// TIA Portal V16 export
// export: Created 2024-08-19T08:04:42.5186365Z, ExportSetting WithDefaults, DisplayName Totally Integrated Automation Portal, DisplayVersion V16, DisplayName TIA Portal Version Control Interface, DisplayVersion V16, DisplayName TIA Portal Openness, DisplayVersion V16, DisplayName STEP 7 Professional, DisplayVersion V16, DisplayName STEP 7 Safety, DisplayVersion V16, DisplayName WinCC Professional, DisplayVersion V16
DATA_BLOCK "DB00801_St_ConstAiRawData"   // DB801
TITLE = Static DB [SYSTEM CONSTANTS] — Analog Input Card Types, Ranges and Coefficients
{ S7_Optimized_Access := 'TRUE' }
AUTHOR : M_Gledhill
FAMILY : SysConstants
NAME : St_ConstAiRawData
VERSION : 1.0
// PRACTICAL SERIES AUTOMATION LIBRARY (PAL)   —   COPYRIGHT 2020 – M. GLEDHILL (MIT LICENCE)
//                   ———— ◆ ————
// FULL ONLINE DOCUMENTATION IS AVAILABLE AT: https://practicalseries.com/2001-pal/index.html
// stored: AutoNumber false, DBAccessibleFromOPCUA true, IsOnlyStoredInLoadMemory false, IsRetainMemResEnabled false, IsWriteProtectedInAS false, MemoryReserve 100
   VAR
      _DB_Header { ExternalAccessible := 'False'; ExternalVisible := 'False'; ExternalWritable := 'False'} : Array[0..79] of Bool;   // Static DB [SYSTEM CONSTANTS] — Analog Input Card Types, Ranges and Coefficients
      __________0000_0 { ExternalAccessible := 'False'; ExternalVisible := 'False'; ExternalWritable := 'False'} : Bool := false;
      __________0000_1 { ExternalAccessible := 'False'; ExternalVisible := 'False'; ExternalWritable := 'False'} : Bool := false;
      revInfo { ExternalWritable := 'False'} : "UT01000_St_SysRevision";
      __________0010_0 { ExternalAccessible := 'False'; ExternalVisible := 'False'; ExternalWritable := 'False'} : Bool := false;
      __________0010_1 { ExternalAccessible := 'False'; ExternalVisible := 'False'; ExternalWritable := 'False'} : Bool := false;
      AI_RAW_0000 { ExternalWritable := 'False'} : "UT00801_St_ConstAiRawData";   // AI User defined signal type
      __________0020_0 { ExternalAccessible := 'False'; ExternalVisible := 'False'; ExternalWritable := 'False'} : Bool := false;
      __________0020_1 { ExternalAccessible := 'False'; ExternalVisible := 'False'; ExternalWritable := 'False'} : Bool := false;   // ▀▀▀▀ ANALOG INPUT SIGNAL — VOLTAGE
      AI_RAW_1000 { ExternalWritable := 'False'} : "UT00801_St_ConstAiRawData";   // AI Voltage (-25 mV to +25 mV)
      AI_RAW_1001 { ExternalWritable := 'False'} : "UT00801_St_ConstAiRawData";   // AI Voltage (-50 mV to +50 mV)
      AI_RAW_1002 { ExternalWritable := 'False'} : "UT00801_St_ConstAiRawData";   // AI Voltage (-80 mV to +80 mV)
      AI_RAW_1003 { ExternalWritable := 'False'} : "UT00801_St_ConstAiRawData";   // AI Voltage (-250 mV to +250 mV)
      AI_RAW_1004 { ExternalWritable := 'False'} : "UT00801_St_ConstAiRawData";   // AI Voltage (-500 mV to +500 mV)
      AI_RAW_1005 { ExternalWritable := 'False'} : "UT00801_St_ConstAiRawData";   // AI Voltage (-1 V to +1 V)
      AI_RAW_1007 { ExternalWritable := 'False'} : "UT00801_St_ConstAiRawData";   // AI Voltage (-2.5 V to +2.5 V)
      AI_RAW_1008 { ExternalWritable := 'False'} : "UT00801_St_ConstAiRawData";   // AI Voltage (-5 V to +5 V)
      AI_RAW_1009 { ExternalWritable := 'False'} : "UT00801_St_ConstAiRawData";   // AI Voltage (-10 V to +10 V)
      AI_RAW_100A { ExternalWritable := 'False'} : "UT00801_St_ConstAiRawData";   // AI Voltage (1 V to 5 V)
      __________0030_0 { ExternalAccessible := 'False'; ExternalVisible := 'False'; ExternalWritable := 'False'} : Bool := false;
      __________0030_1 { ExternalAccessible := 'False'; ExternalVisible := 'False'; ExternalWritable := 'False'} : Bool := false;   // ▀▀▀▀ ANALOG INPUT SIGNAL — CURRENT (4 WIRE)
      AI_RAW_2002 { ExternalWritable := 'False'} : "UT00801_St_ConstAiRawData";   // AI Current - 4-wire (0 mA to 20 mA)
      AI_RAW_2003 { ExternalWritable := 'False'} : "UT00801_St_ConstAiRawData";   // AI Current - 4-wire (4 mA to 20 mA)
      AI_RAW_2004 { ExternalWritable := 'False'} : "UT00801_St_ConstAiRawData";   // AI Current - 4-wire (-20 mA to +20 mA)
      __________0040_0 { ExternalAccessible := 'False'; ExternalVisible := 'False'; ExternalWritable := 'False'} : Bool := false;
      __________0040_1 { ExternalAccessible := 'False'; ExternalVisible := 'False'; ExternalWritable := 'False'} : Bool := false;   // ▀▀▀▀ ANALOG INPUT SIGNAL — CURRENT (2 WIRE)
      AI_RAW_3003 { ExternalWritable := 'False'} : "UT00801_St_ConstAiRawData";   // AI Current - 2-wire (4 mA to 20 mA)
      __________0050_0 { ExternalAccessible := 'False'; ExternalVisible := 'False'; ExternalWritable := 'False'} : Bool := false;
      __________0050_1 { ExternalAccessible := 'False'; ExternalVisible := 'False'; ExternalWritable := 'False'} : Bool := false;   // ▀▀▀▀ ANALOG INPUT SIGNAL — RESISTANCE (4 WIRE)
      AI_RAW_4001 { ExternalWritable := 'False'} : "UT00801_St_ConstAiRawData";   // AI Resistance - 4-wire (150 Ohm)
      AI_RAW_4002 { ExternalWritable := 'False'} : "UT00801_St_ConstAiRawData";   // AI Resistance - 4-wire (300 Ohm)
      AI_RAW_4003 { ExternalWritable := 'False'} : "UT00801_St_ConstAiRawData";   // AI Resistance - 4-wire (600 Ohm)
      AI_RAW_4005 { ExternalWritable := 'False'} : "UT00801_St_ConstAiRawData";   // AI Resistance - 4-wire (6000 Ohm)
      __________0060_0 { ExternalAccessible := 'False'; ExternalVisible := 'False'; ExternalWritable := 'False'} : Bool := false;
      __________0060_1 { ExternalAccessible := 'False'; ExternalVisible := 'False'; ExternalWritable := 'False'} : Bool := false;   // ▀▀▀▀ ANALOG INPUT SIGNAL — RESISTANCE (3 WIRE)
      AI_RAW_5001 { ExternalWritable := 'False'} : "UT00801_St_ConstAiRawData";   // AI Resistance - 3-wire (150 Ohm)
      AI_RAW_5002 { ExternalWritable := 'False'} : "UT00801_St_ConstAiRawData";   // AI Resistance - 3-wire (300 Ohm)
      AI_RAW_5003 { ExternalWritable := 'False'} : "UT00801_St_ConstAiRawData";   // AI Resistance - 3-wire (600 Ohm)
      AI_RAW_5005 { ExternalWritable := 'False'} : "UT00801_St_ConstAiRawData";   // AI Resistance - 3-wire (6000 Ohm)
      __________0070_0 { ExternalAccessible := 'False'; ExternalVisible := 'False'; ExternalWritable := 'False'} : Bool := false;
      __________0070_1 { ExternalAccessible := 'False'; ExternalVisible := 'False'; ExternalWritable := 'False'} : Bool := false;   // ▀▀▀▀ ANALOG INPUT SIGNAL — RESISTANCE (2 WIRE)
      AI_RAW_6001 { ExternalWritable := 'False'} : "UT00801_St_ConstAiRawData";   // AI Resistance - 2-wire (150 Ohm)
      AI_RAW_6002 { ExternalWritable := 'False'} : "UT00801_St_ConstAiRawData";   // AI Resistance - 2-wire (300 Ohm)
      AI_RAW_6003 { ExternalWritable := 'False'} : "UT00801_St_ConstAiRawData";   // AI Resistance - 2-wire (600 Ohm)
      AI_RAW_6005 { ExternalWritable := 'False'} : "UT00801_St_ConstAiRawData";   // AI Resistance - 2-wire (6000 Ohm)
      AI_RAW_600F { ExternalWritable := 'False'} : "UT00801_St_ConstAiRawData";   // AI Resistance - 2-wire (PTC)
      __________0080_0 { ExternalAccessible := 'False'; ExternalVisible := 'False'; ExternalWritable := 'False'} : Bool := false;
      __________0080_1 { ExternalAccessible := 'False'; ExternalVisible := 'False'; ExternalWritable := 'False'} : Bool := false;   // ▀▀▀▀ ANALOG INPUT SIGNAL — THERMAL RESISTANCE (4 WIRE) Cu x0
      AI_RAW_7B0E { ExternalWritable := 'False'} : "UT00801_St_ConstAiRawData";   // AI Thermal Resistance - 4-wire (Cu10 climate - 426)
      AI_RAW_7C0E { ExternalWritable := 'False'} : "UT00801_St_ConstAiRawData";   // AI Thermal Resistance - 4-wire (Cu10 climate - 427)
      AI_RAW_7D0E { ExternalWritable := 'False'} : "UT00801_St_ConstAiRawData";   // AI Thermal Resistance - 4-wire (Cu10 climate - 428)
      AI_RAW_7B0F { ExternalWritable := 'False'} : "UT00801_St_ConstAiRawData";   // AI Thermal Resistance - 4-wire (Cu10 standard - 426)
      AI_RAW_7C0F { ExternalWritable := 'False'} : "UT00801_St_ConstAiRawData";   // AI Thermal Resistance - 4-wire (Cu10 standard - 427)
      AI_RAW_7D0F { ExternalWritable := 'False'} : "UT00801_St_ConstAiRawData";   // AI Thermal Resistance - 4-wire (Cu10 standard - 428)
      AI_RAW_7B19 { ExternalWritable := 'False'} : "UT00801_St_ConstAiRawData";   // AI Thermal Resistance - 4-wire (Cu50 climate - 426)
      AI_RAW_7C19 { ExternalWritable := 'False'} : "UT00801_St_ConstAiRawData";   // AI Thermal Resistance - 4-wire (Cu50 climate - 427)
      AI_RAW_7D19 { ExternalWritable := 'False'} : "UT00801_St_ConstAiRawData";   // AI Thermal Resistance - 4-wire (Cu50 climate - 428)
      AI_RAW_7B18 { ExternalWritable := 'False'} : "UT00801_St_ConstAiRawData";   // AI Thermal Resistance - 4-wire (Cu50 standard - 426)
      AI_RAW_7C18 { ExternalWritable := 'False'} : "UT00801_St_ConstAiRawData";   // AI Thermal Resistance - 4-wire (Cu50 standard - 427)
      AI_RAW_7D18 { ExternalWritable := 'False'} : "UT00801_St_ConstAiRawData";   // AI Thermal Resistance - 4-wire (Cu50 standard - 428)
      AI_RAW_7B1B { ExternalWritable := 'False'} : "UT00801_St_ConstAiRawData";   // AI Thermal Resistance - 4-wire (Cu100 climate - 426)
      AI_RAW_7C1B { ExternalWritable := 'False'} : "UT00801_St_ConstAiRawData";   // AI Thermal Resistance - 4-wire (Cu100 climate - 427)
      AI_RAW_7D1B { ExternalWritable := 'False'} : "UT00801_St_ConstAiRawData";   // AI Thermal Resistance - 4-wire (Cu100 climate - 428)
      AI_RAW_7B1A { ExternalWritable := 'False'} : "UT00801_St_ConstAiRawData";   // AI Thermal Resistance - 4-wire (Cu100 standard - 426)
      AI_RAW_7C1A { ExternalWritable := 'False'} : "UT00801_St_ConstAiRawData";   // AI Thermal Resistance - 4-wire (Cu100 standard - 427)
      AI_RAW_7D1A { ExternalWritable := 'False'} : "UT00801_St_ConstAiRawData";   // AI Thermal Resistance - 4-wire (Cu100 standard - 428)
      __________0090_0 { ExternalAccessible := 'False'; ExternalVisible := 'False'; ExternalWritable := 'False'} : Bool := false;
      __________0090_1 { ExternalAccessible := 'False'; ExternalVisible := 'False'; ExternalWritable := 'False'} : Bool := false;   // ▀▀▀▀ ANALOG INPUT SIGNAL — THERMAL RESISTANCE (4 WIRE) LG-Ni x0
      AI_RAW_7A1D { ExternalWritable := 'False'} : "UT00801_St_ConstAiRawData";   // AI Thermal Resistance - 4-wire (LG-Ni1000 climate - 500)
      AI_RAW_7A1C { ExternalWritable := 'False'} : "UT00801_St_ConstAiRawData";   // AI Thermal Resistance - 4-wire (LG-Ni1000 standard - 500)
      __________0100_0 { ExternalAccessible := 'False'; ExternalVisible := 'False'; ExternalWritable := 'False'} : Bool := false;
      __________0100_1 { ExternalAccessible := 'False'; ExternalVisible := 'False'; ExternalWritable := 'False'} : Bool := false;   // ▀▀▀▀ ANALOG INPUT SIGNAL — THERMAL RESISTANCE (4 WIRE) Ni x0
      AI_RAW_771F { ExternalWritable := 'False'} : "UT00801_St_ConstAiRawData";   // AI Thermal Resistance - 4-wire (Ni10 climate - 617)
      AI_RAW_781F { ExternalWritable := 'False'} : "UT00801_St_ConstAiRawData";   // AI Thermal Resistance - 4-wire (Ni10 climate - 618)
      AI_RAW_791F { ExternalWritable := 'False'} : "UT00801_St_ConstAiRawData";   // AI Thermal Resistance - 4-wire (Ni10 climate - 672)
      AI_RAW_771E { ExternalWritable := 'False'} : "UT00801_St_ConstAiRawData";   // AI Thermal Resistance - 4-wire (Ni10 standard - 617)
      AI_RAW_781E { ExternalWritable := 'False'} : "UT00801_St_ConstAiRawData";   // AI Thermal Resistance - 4-wire (Ni10 standard - 618)
      AI_RAW_791E { ExternalWritable := 'False'} : "UT00801_St_ConstAiRawData";   // AI Thermal Resistance - 4-wire (Ni10 standard - 672)
      AI_RAW_770D { ExternalWritable := 'False'} : "UT00801_St_ConstAiRawData";   // AI Thermal Resistance - 4-wire (Ni120 climate - 617)
      AI_RAW_780D { ExternalWritable := 'False'} : "UT00801_St_ConstAiRawData";   // AI Thermal Resistance - 4-wire (Ni120 climate - 618)
      AI_RAW_790D { ExternalWritable := 'False'} : "UT00801_St_ConstAiRawData";   // AI Thermal Resistance - 4-wire (Ni120 climate - 672)
      AI_RAW_770C { ExternalWritable := 'False'} : "UT00801_St_ConstAiRawData";   // AI Thermal Resistance - 4-wire (Ni120 standard - 617)
      AI_RAW_780C { ExternalWritable := 'False'} : "UT00801_St_ConstAiRawData";   // AI Thermal Resistance - 4-wire (Ni120 standard - 618)
      AI_RAW_790C { ExternalWritable := 'False'} : "UT00801_St_ConstAiRawData";   // AI Thermal Resistance - 4-wire (Ni120 standard - 672)
      AI_RAW_7701 { ExternalWritable := 'False'} : "UT00801_St_ConstAiRawData";   // AI Thermal Resistance - 4-wire (Ni100 climate - 617)
      AI_RAW_7801 { ExternalWritable := 'False'} : "UT00801_St_ConstAiRawData";   // AI Thermal Resistance - 4-wire (Ni100 climate - 618)
      AI_RAW_7901 { ExternalWritable := 'False'} : "UT00801_St_ConstAiRawData";   // AI Thermal Resistance - 4-wire (Ni100 climate - 672)
      AI_RAW_7703 { ExternalWritable := 'False'} : "UT00801_St_ConstAiRawData";   // AI Thermal Resistance - 4-wire (Ni100 standard - 617)
      AI_RAW_7803 { ExternalWritable := 'False'} : "UT00801_St_ConstAiRawData";   // AI Thermal Resistance - 4-wire (Ni100 standard - 618)
      AI_RAW_7903 { ExternalWritable := 'False'} : "UT00801_St_ConstAiRawData";   // AI Thermal Resistance - 4-wire (Ni100 standard - 672)
      AI_RAW_7711 { ExternalWritable := 'False'} : "UT00801_St_ConstAiRawData";   // AI Thermal Resistance - 4-wire (Ni200 climate - 617)
      AI_RAW_7811 { ExternalWritable := 'False'} : "UT00801_St_ConstAiRawData";   // AI Thermal Resistance - 4-wire (Ni200 climate - 618)
      AI_RAW_7911 { ExternalWritable := 'False'} : "UT00801_St_ConstAiRawData";   // AI Thermal Resistance - 4-wire (Ni200 climate - 672)
      AI_RAW_7710 { ExternalWritable := 'False'} : "UT00801_St_ConstAiRawData";   // AI Thermal Resistance - 4-wire (Ni200 standard - 617)
      AI_RAW_7810 { ExternalWritable := 'False'} : "UT00801_St_ConstAiRawData";   // AI Thermal Resistance - 4-wire (Ni200 standard - 618)
      AI_RAW_7910 { ExternalWritable := 'False'} : "UT00801_St_ConstAiRawData";   // AI Thermal Resistance - 4-wire (Ni200 standard - 672)
      AI_RAW_7713 { ExternalWritable := 'False'} : "UT00801_St_ConstAiRawData";   // AI Thermal Resistance - 4-wire (Ni500 climate - 617)
      AI_RAW_7813 { ExternalWritable := 'False'} : "UT00801_St_ConstAiRawData";   // AI Thermal Resistance - 4-wire (Ni500 climate - 618)
      AI_RAW_7913 { ExternalWritable := 'False'} : "UT00801_St_ConstAiRawData";   // AI Thermal Resistance - 4-wire (Ni500 climate - 672)
      AI_RAW_7712 { ExternalWritable := 'False'} : "UT00801_St_ConstAiRawData";   // AI Thermal Resistance - 4-wire (Ni500 standard - 617)
      AI_RAW_7812 { ExternalWritable := 'False'} : "UT00801_St_ConstAiRawData";   // AI Thermal Resistance - 4-wire (Ni500 standard - 618)
      AI_RAW_7912 { ExternalWritable := 'False'} : "UT00801_St_ConstAiRawData";   // AI Thermal Resistance - 4-wire (Ni500 standard - 672)
      AI_RAW_770A { ExternalWritable := 'False'} : "UT00801_St_ConstAiRawData";   // AI Thermal Resistance - 4-wire (Ni1000 climate - 617)
      AI_RAW_780A { ExternalWritable := 'False'} : "UT00801_St_ConstAiRawData";   // AI Thermal Resistance - 4-wire (Ni1000 climate - 618)
      AI_RAW_790A { ExternalWritable := 'False'} : "UT00801_St_ConstAiRawData";   // AI Thermal Resistance - 4-wire (Ni1000 climate - 672)
      AI_RAW_7706 { ExternalWritable := 'False'} : "UT00801_St_ConstAiRawData";   // AI Thermal Resistance - 4-wire (Ni1000 standard - 617)
      AI_RAW_7806 { ExternalWritable := 'False'} : "UT00801_St_ConstAiRawData";   // AI Thermal Resistance - 4-wire (Ni1000 standard - 618)
      AI_RAW_7906 { ExternalWritable := 'False'} : "UT00801_St_ConstAiRawData";   // AI Thermal Resistance - 4-wire (Ni1000 standard - 672)
      __________0110_0 { ExternalAccessible := 'False'; ExternalVisible := 'False'; ExternalWritable := 'False'} : Bool := false;
      __________0110_1 { ExternalAccessible := 'False'; ExternalVisible := 'False'; ExternalWritable := 'False'} : Bool := false;   // ▀▀▀▀ ANALOG INPUT SIGNAL — THERMAL RESISTANCE (4 WIRE) Pt x0
      AI_RAW_7015 { ExternalWritable := 'False'} : "UT00801_St_ConstAiRawData";   // AI Thermal Resistance - 4-wire (Pt10 climate - 3851)
      AI_RAW_7215 { ExternalWritable := 'False'} : "UT00801_St_ConstAiRawData";   // AI Thermal Resistance - 4-wire (Pt10 climate - 3902)
      AI_RAW_7515 { ExternalWritable := 'False'} : "UT00801_St_ConstAiRawData";   // AI Thermal Resistance - 4-wire (Pt10 climate - 391)
      AI_RAW_7115 { ExternalWritable := 'False'} : "UT00801_St_ConstAiRawData";   // AI Thermal Resistance - 4-wire (Pt10 climate - 3916)
      AI_RAW_7315 { ExternalWritable := 'False'} : "UT00801_St_ConstAiRawData";   // AI Thermal Resistance - 4-wire (Pt10 climate - 392)
      AI_RAW_7014 { ExternalWritable := 'False'} : "UT00801_St_ConstAiRawData";   // AI Thermal Resistance - 4-wire (Pt10 standard - 3851)
      AI_RAW_7214 { ExternalWritable := 'False'} : "UT00801_St_ConstAiRawData";   // AI Thermal Resistance - 4-wire (Pt10 standard - 3902)
      AI_RAW_7514 { ExternalWritable := 'False'} : "UT00801_St_ConstAiRawData";   // AI Thermal Resistance - 4-wire (Pt10 standard - 391)
      AI_RAW_7114 { ExternalWritable := 'False'} : "UT00801_St_ConstAiRawData";   // AI Thermal Resistance - 4-wire (Pt10 standard - 3916)
      AI_RAW_7314 { ExternalWritable := 'False'} : "UT00801_St_ConstAiRawData";   // AI Thermal Resistance - 4-wire (Pt10 standard - 392)
      AI_RAW_7017 { ExternalWritable := 'False'} : "UT00801_St_ConstAiRawData";   // AI Thermal Resistance - 4-wire (Pt50 climate - 3851)
      AI_RAW_7217 { ExternalWritable := 'False'} : "UT00801_St_ConstAiRawData";   // AI Thermal Resistance - 4-wire (Pt50 climate - 3902)
      AI_RAW_7517 { ExternalWritable := 'False'} : "UT00801_St_ConstAiRawData";   // AI Thermal Resistance - 4-wire (Pt50 climate - 391)
      AI_RAW_7117 { ExternalWritable := 'False'} : "UT00801_St_ConstAiRawData";   // AI Thermal Resistance - 4-wire (Pt50 climate - 3916)
      AI_RAW_7317 { ExternalWritable := 'False'} : "UT00801_St_ConstAiRawData";   // AI Thermal Resistance - 4-wire (Pt50 climate - 392)
      AI_RAW_7016 { ExternalWritable := 'False'} : "UT00801_St_ConstAiRawData";   // AI Thermal Resistance - 4-wire (Pt50 standard - 3851)
      AI_RAW_7216 { ExternalWritable := 'False'} : "UT00801_St_ConstAiRawData";   // AI Thermal Resistance - 4-wire (Pt50 standard - 3902)
      AI_RAW_7516 { ExternalWritable := 'False'} : "UT00801_St_ConstAiRawData";   // AI Thermal Resistance - 4-wire (Pt50 standard - 391)
      AI_RAW_7116 { ExternalWritable := 'False'} : "UT00801_St_ConstAiRawData";   // AI Thermal Resistance - 4-wire (Pt50 standard - 3916)
      AI_RAW_7316 { ExternalWritable := 'False'} : "UT00801_St_ConstAiRawData";   // AI Thermal Resistance - 4-wire (Pt50 standard - 392)
      AI_RAW_7000 { ExternalWritable := 'False'} : "UT00801_St_ConstAiRawData";   // AI Thermal Resistance - 4-wire (Pt100 climate - 3851)
      AI_RAW_7200 { ExternalWritable := 'False'} : "UT00801_St_ConstAiRawData";   // AI Thermal Resistance - 4-wire (Pt100 climate - 3902)
      AI_RAW_7500 { ExternalWritable := 'False'} : "UT00801_St_ConstAiRawData";   // AI Thermal Resistance - 4-wire (Pt100 climate - 391)
      AI_RAW_7100 { ExternalWritable := 'False'} : "UT00801_St_ConstAiRawData";   // AI Thermal Resistance - 4-wire (Pt100 climate - 3916)
      AI_RAW_7300 { ExternalWritable := 'False'} : "UT00801_St_ConstAiRawData";   // AI Thermal Resistance - 4-wire (Pt100 climate - 392)
      AI_RAW_7002 { ExternalWritable := 'False'} : "UT00801_St_ConstAiRawData";   // AI Thermal Resistance - 4-wire (Pt100 standard - 3851)
      AI_RAW_7202 { ExternalWritable := 'False'} : "UT00801_St_ConstAiRawData";   // AI Thermal Resistance - 4-wire (Pt100 standard - 3902)
      AI_RAW_7502 { ExternalWritable := 'False'} : "UT00801_St_ConstAiRawData";   // AI Thermal Resistance - 4-wire (Pt100 standard - 391)
      AI_RAW_7102 { ExternalWritable := 'False'} : "UT00801_St_ConstAiRawData";   // AI Thermal Resistance - 4-wire (Pt100 standard - 3916)
      AI_RAW_7302 { ExternalWritable := 'False'} : "UT00801_St_ConstAiRawData";   // AI Thermal Resistance - 4-wire (Pt100 standard - 392)
      AI_RAW_7007 { ExternalWritable := 'False'} : "UT00801_St_ConstAiRawData";   // AI Thermal Resistance - 4-wire (Pt200 climate - 3851)
      AI_RAW_7207 { ExternalWritable := 'False'} : "UT00801_St_ConstAiRawData";   // AI Thermal Resistance - 4-wire (Pt200 climate - 3902)
      AI_RAW_7507 { ExternalWritable := 'False'} : "UT00801_St_ConstAiRawData";   // AI Thermal Resistance - 4-wire (Pt200 climate - 391)
      AI_RAW_7107 { ExternalWritable := 'False'} : "UT00801_St_ConstAiRawData";   // AI Thermal Resistance - 4-wire (Pt200 climate - 3916)
      AI_RAW_7307 { ExternalWritable := 'False'} : "UT00801_St_ConstAiRawData";   // AI Thermal Resistance - 4-wire (Pt200 climate - 392)
      AI_RAW_700B { ExternalWritable := 'False'} : "UT00801_St_ConstAiRawData";   // AI Thermal Resistance - 4-wire (Pt200 standard - 3851)
      AI_RAW_720B { ExternalWritable := 'False'} : "UT00801_St_ConstAiRawData";   // AI Thermal Resistance - 4-wire (Pt200 standard - 3902)
      AI_RAW_750B { ExternalWritable := 'False'} : "UT00801_St_ConstAiRawData";   // AI Thermal Resistance - 4-wire (Pt200 standard - 391)
      AI_RAW_710B { ExternalWritable := 'False'} : "UT00801_St_ConstAiRawData";   // AI Thermal Resistance - 4-wire (Pt200 standard - 3916)
      AI_RAW_730B { ExternalWritable := 'False'} : "UT00801_St_ConstAiRawData";   // AI Thermal Resistance - 4-wire (Pt200 standard - 392)
      AI_RAW_7008 { ExternalWritable := 'False'} : "UT00801_St_ConstAiRawData";   // AI Thermal Resistance - 4-wire (Pt500 climate - 3851)
      AI_RAW_7208 { ExternalWritable := 'False'} : "UT00801_St_ConstAiRawData";   // AI Thermal Resistance - 4-wire (Pt500 climate - 3902)
      AI_RAW_7508 { ExternalWritable := 'False'} : "UT00801_St_ConstAiRawData";   // AI Thermal Resistance - 4-wire (Pt500 climate - 391)
      AI_RAW_7108 { ExternalWritable := 'False'} : "UT00801_St_ConstAiRawData";   // AI Thermal Resistance - 4-wire (Pt500 climate - 3916)
      AI_RAW_7308 { ExternalWritable := 'False'} : "UT00801_St_ConstAiRawData";   // AI Thermal Resistance - 4-wire (Pt500 climate - 392)
      AI_RAW_7004 { ExternalWritable := 'False'} : "UT00801_St_ConstAiRawData";   // AI Thermal Resistance - 4-wire (Pt500 standard - 3851)
      AI_RAW_7204 { ExternalWritable := 'False'} : "UT00801_St_ConstAiRawData";   // AI Thermal Resistance - 4-wire (Pt500 standard - 3902)
      AI_RAW_7504 { ExternalWritable := 'False'} : "UT00801_St_ConstAiRawData";   // AI Thermal Resistance - 4-wire (Pt500 standard - 391)
      AI_RAW_7104 { ExternalWritable := 'False'} : "UT00801_St_ConstAiRawData";   // AI Thermal Resistance - 4-wire (Pt500 standard - 3916)
      AI_RAW_7304 { ExternalWritable := 'False'} : "UT00801_St_ConstAiRawData";   // AI Thermal Resistance - 4-wire (Pt500 standard - 392)
      AI_RAW_7009 { ExternalWritable := 'False'} : "UT00801_St_ConstAiRawData";   // AI Thermal Resistance - 4-wire (Pt1000 climate - 3851)
      AI_RAW_7209 { ExternalWritable := 'False'} : "UT00801_St_ConstAiRawData";   // AI Thermal Resistance - 4-wire (Pt1000 climate - 3902)
      AI_RAW_7509 { ExternalWritable := 'False'} : "UT00801_St_ConstAiRawData";   // AI Thermal Resistance - 4-wire (Pt1000 climate - 391)
      AI_RAW_7109 { ExternalWritable := 'False'} : "UT00801_St_ConstAiRawData";   // AI Thermal Resistance - 4-wire (Pt1000 climate - 3916)
      AI_RAW_7309 { ExternalWritable := 'False'} : "UT00801_St_ConstAiRawData";   // AI Thermal Resistance - 4-wire (Pt1000 climate - 392)
      AI_RAW_7005 { ExternalWritable := 'False'} : "UT00801_St_ConstAiRawData";   // AI Thermal Resistance - 4-wire (Pt1000 standard - 3851)
      AI_RAW_7205 { ExternalWritable := 'False'} : "UT00801_St_ConstAiRawData";   // AI Thermal Resistance - 4-wire (Pt1000 standard - 3902)
      AI_RAW_7505 { ExternalWritable := 'False'} : "UT00801_St_ConstAiRawData";   // AI Thermal Resistance - 4-wire (Pt1000 standard - 391)
      AI_RAW_7105 { ExternalWritable := 'False'} : "UT00801_St_ConstAiRawData";   // AI Thermal Resistance - 4-wire (Pt1000 standard - 3916)
      AI_RAW_7305 { ExternalWritable := 'False'} : "UT00801_St_ConstAiRawData";   // AI Thermal Resistance - 4-wire (Pt1000 standard - 392)
      __________0120_0 { ExternalAccessible := 'False'; ExternalVisible := 'False'; ExternalWritable := 'False'} : Bool := false;
      __________0120_1 { ExternalAccessible := 'False'; ExternalVisible := 'False'; ExternalWritable := 'False'} : Bool := false;   // ▀▀▀▀ ANALOG INPUT SIGNAL — THERMAL RESISTANCE (3 WIRE) Cu x0
      AI_RAW_8B0E { ExternalWritable := 'False'} : "UT00801_St_ConstAiRawData";   // AI Thermal Resistance - 3-wire (Cu10 climate - 426)
      AI_RAW_8C0E { ExternalWritable := 'False'} : "UT00801_St_ConstAiRawData";   // AI Thermal Resistance - 3-wire (Cu10 climate - 427)
      AI_RAW_8D0E { ExternalWritable := 'False'} : "UT00801_St_ConstAiRawData";   // AI Thermal Resistance - 3-wire (Cu10 climate - 428)
      AI_RAW_8B0F { ExternalWritable := 'False'} : "UT00801_St_ConstAiRawData";   // AI Thermal Resistance - 3-wire (Cu10 standard - 426)
      AI_RAW_8C0F { ExternalWritable := 'False'} : "UT00801_St_ConstAiRawData";   // AI Thermal Resistance - 3-wire (Cu10 standard - 427)
      AI_RAW_8D0F { ExternalWritable := 'False'} : "UT00801_St_ConstAiRawData";   // AI Thermal Resistance - 3-wire (Cu10 standard - 428)
      AI_RAW_8B19 { ExternalWritable := 'False'} : "UT00801_St_ConstAiRawData";   // AI Thermal Resistance - 3-wire (Cu50 climate - 426)
      AI_RAW_8C19 { ExternalWritable := 'False'} : "UT00801_St_ConstAiRawData";   // AI Thermal Resistance - 3-wire (Cu50 climate - 427)
      AI_RAW_8D19 { ExternalWritable := 'False'} : "UT00801_St_ConstAiRawData";   // AI Thermal Resistance - 3-wire (Cu50 climate - 428)
      AI_RAW_8B18 { ExternalWritable := 'False'} : "UT00801_St_ConstAiRawData";   // AI Thermal Resistance - 3-wire (Cu50 standard - 426)
      AI_RAW_8C18 { ExternalWritable := 'False'} : "UT00801_St_ConstAiRawData";   // AI Thermal Resistance - 3-wire (Cu50 standard - 427)
      AI_RAW_8D18 { ExternalWritable := 'False'} : "UT00801_St_ConstAiRawData";   // AI Thermal Resistance - 3-wire (Cu50 standard - 428)
      AI_RAW_8B1B { ExternalWritable := 'False'} : "UT00801_St_ConstAiRawData";   // AI Thermal Resistance - 3-wire (Cu100 climate - 426)
      AI_RAW_8C1B { ExternalWritable := 'False'} : "UT00801_St_ConstAiRawData";   // AI Thermal Resistance - 3-wire (Cu100 climate - 427)
      AI_RAW_8D1B { ExternalWritable := 'False'} : "UT00801_St_ConstAiRawData";   // AI Thermal Resistance - 3-wire (Cu100 climate - 428)
      AI_RAW_8B1A { ExternalWritable := 'False'} : "UT00801_St_ConstAiRawData";   // AI Thermal Resistance - 3-wire (Cu100 standard - 426)
      AI_RAW_8C1A { ExternalWritable := 'False'} : "UT00801_St_ConstAiRawData";   // AI Thermal Resistance - 3-wire (Cu100 standard - 427)
      AI_RAW_8D1A { ExternalWritable := 'False'} : "UT00801_St_ConstAiRawData";   // AI Thermal Resistance - 3-wire (Cu100 standard - 428)
      __________0130_0 { ExternalAccessible := 'False'; ExternalVisible := 'False'; ExternalWritable := 'False'} : Bool := false;
      __________0130_1 { ExternalAccessible := 'False'; ExternalVisible := 'False'; ExternalWritable := 'False'} : Bool := false;   // ▀▀▀▀ ANALOG INPUT SIGNAL — THERMAL RESISTANCE (3 WIRE) LG-Ni x0
      AI_RAW_8A1D { ExternalWritable := 'False'} : "UT00801_St_ConstAiRawData";   // AI Thermal Resistance - 3-wire (LG-Ni1000 climate - 500)
      AI_RAW_8A1C { ExternalWritable := 'False'} : "UT00801_St_ConstAiRawData";   // AI Thermal Resistance - 3-wire (LG-Ni1000 standard - 500)
      __________0140_0 { ExternalAccessible := 'False'; ExternalVisible := 'False'; ExternalWritable := 'False'} : Bool := false;
      __________0140_1 { ExternalAccessible := 'False'; ExternalVisible := 'False'; ExternalWritable := 'False'} : Bool := false;   // ▀▀▀▀ ANALOG INPUT SIGNAL — THERMAL RESISTANCE (3 WIRE) Ni x0
      AI_RAW_871F { ExternalWritable := 'False'} : "UT00801_St_ConstAiRawData";   // AI Thermal Resistance - 3-wire (Ni10 climate - 617)
      AI_RAW_881F { ExternalWritable := 'False'} : "UT00801_St_ConstAiRawData";   // AI Thermal Resistance - 3-wire (Ni10 climate - 618)
      AI_RAW_891F { ExternalWritable := 'False'} : "UT00801_St_ConstAiRawData";   // AI Thermal Resistance - 3-wire (Ni10 climate - 672)
      AI_RAW_871E { ExternalWritable := 'False'} : "UT00801_St_ConstAiRawData";   // AI Thermal Resistance - 3-wire (Ni10 standard - 617)
      AI_RAW_881E { ExternalWritable := 'False'} : "UT00801_St_ConstAiRawData";   // AI Thermal Resistance - 3-wire (Ni10 standard - 618)
      AI_RAW_891E { ExternalWritable := 'False'} : "UT00801_St_ConstAiRawData";   // AI Thermal Resistance - 3-wire (Ni10 standard - 672)
      AI_RAW_870D { ExternalWritable := 'False'} : "UT00801_St_ConstAiRawData";   // AI Thermal Resistance - 3-wire (Ni120 climate - 617)
      AI_RAW_880D { ExternalWritable := 'False'} : "UT00801_St_ConstAiRawData";   // AI Thermal Resistance - 3-wire (Ni120 climate - 618)
      AI_RAW_890D { ExternalWritable := 'False'} : "UT00801_St_ConstAiRawData";   // AI Thermal Resistance - 3-wire (Ni120 climate - 672)
      AI_RAW_870C { ExternalWritable := 'False'} : "UT00801_St_ConstAiRawData";   // AI Thermal Resistance - 3-wire (Ni120 standard - 617)
      AI_RAW_880C { ExternalWritable := 'False'} : "UT00801_St_ConstAiRawData";   // AI Thermal Resistance - 3-wire (Ni120 standard - 618)
      AI_RAW_890C { ExternalWritable := 'False'} : "UT00801_St_ConstAiRawData";   // AI Thermal Resistance - 3-wire (Ni120 standard - 672)
      AI_RAW_8701 { ExternalWritable := 'False'} : "UT00801_St_ConstAiRawData";   // AI Thermal Resistance - 3-wire (Ni100 climate - 617)
      AI_RAW_8801 { ExternalWritable := 'False'} : "UT00801_St_ConstAiRawData";   // AI Thermal Resistance - 3-wire (Ni100 climate - 618)
      AI_RAW_8901 { ExternalWritable := 'False'} : "UT00801_St_ConstAiRawData";   // AI Thermal Resistance - 3-wire (Ni100 climate - 672)
      AI_RAW_8703 { ExternalWritable := 'False'} : "UT00801_St_ConstAiRawData";   // AI Thermal Resistance - 3-wire (Ni100 standard - 617)
      AI_RAW_8803 { ExternalWritable := 'False'} : "UT00801_St_ConstAiRawData";   // AI Thermal Resistance - 3-wire (Ni100 standard - 618)
      AI_RAW_8903 { ExternalWritable := 'False'} : "UT00801_St_ConstAiRawData";   // AI Thermal Resistance - 3-wire (Ni100 standard - 672)
      AI_RAW_8711 { ExternalWritable := 'False'} : "UT00801_St_ConstAiRawData";   // AI Thermal Resistance - 3-wire (Ni200 climate - 617)
      AI_RAW_8811 { ExternalWritable := 'False'} : "UT00801_St_ConstAiRawData";   // AI Thermal Resistance - 3-wire (Ni200 climate - 618)
      AI_RAW_8911 { ExternalWritable := 'False'} : "UT00801_St_ConstAiRawData";   // AI Thermal Resistance - 3-wire (Ni200 climate - 672)
      AI_RAW_8710 { ExternalWritable := 'False'} : "UT00801_St_ConstAiRawData";   // AI Thermal Resistance - 3-wire (Ni200 standard - 617)
      AI_RAW_8810 { ExternalWritable := 'False'} : "UT00801_St_ConstAiRawData";   // AI Thermal Resistance - 3-wire (Ni200 standard - 618)
      AI_RAW_8910 { ExternalWritable := 'False'} : "UT00801_St_ConstAiRawData";   // AI Thermal Resistance - 3-wire (Ni200 standard - 672)
      AI_RAW_8713 { ExternalWritable := 'False'} : "UT00801_St_ConstAiRawData";   // AI Thermal Resistance - 3-wire (Ni500 climate - 617)
      AI_RAW_8813 { ExternalWritable := 'False'} : "UT00801_St_ConstAiRawData";   // AI Thermal Resistance - 3-wire (Ni500 climate - 618)
      AI_RAW_8913 { ExternalWritable := 'False'} : "UT00801_St_ConstAiRawData";   // AI Thermal Resistance - 3-wire (Ni500 climate - 672)
      AI_RAW_8712 { ExternalWritable := 'False'} : "UT00801_St_ConstAiRawData";   // AI Thermal Resistance - 3-wire (Ni500 standard - 617)
      AI_RAW_8812 { ExternalWritable := 'False'} : "UT00801_St_ConstAiRawData";   // AI Thermal Resistance - 3-wire (Ni500 standard - 618)
      AI_RAW_8912 { ExternalWritable := 'False'} : "UT00801_St_ConstAiRawData";   // AI Thermal Resistance - 3-wire (Ni500 standard - 672)
      AI_RAW_870A { ExternalWritable := 'False'} : "UT00801_St_ConstAiRawData";   // AI Thermal Resistance - 3-wire (Ni1000 climate - 617)
      AI_RAW_880A { ExternalWritable := 'False'} : "UT00801_St_ConstAiRawData";   // AI Thermal Resistance - 3-wire (Ni1000 climate - 618)
      AI_RAW_890A { ExternalWritable := 'False'} : "UT00801_St_ConstAiRawData";   // AI Thermal Resistance - 3-wire (Ni1000 climate - 672)
      AI_RAW_8706 { ExternalWritable := 'False'} : "UT00801_St_ConstAiRawData";   // AI Thermal Resistance - 3-wire (Ni1000 standard - 617)
      AI_RAW_8806 { ExternalWritable := 'False'} : "UT00801_St_ConstAiRawData";   // AI Thermal Resistance - 3-wire (Ni1000 standard - 618)
      AI_RAW_8906 { ExternalWritable := 'False'} : "UT00801_St_ConstAiRawData";   // AI Thermal Resistance - 3-wire (Ni1000 standard - 672)
      __________0150_0 { ExternalAccessible := 'False'; ExternalVisible := 'False'; ExternalWritable := 'False'} : Bool := false;
      __________0150_1 { ExternalAccessible := 'False'; ExternalVisible := 'False'; ExternalWritable := 'False'} : Bool := false;   // ▀▀▀▀ ANALOG INPUT SIGNAL — THERMAL RESISTANCE (3 WIRE) Pt x0
      AI_RAW_8015 { ExternalWritable := 'False'} : "UT00801_St_ConstAiRawData";   // AI Thermal Resistance - 3-wire (Pt10 climate - 3851)
      AI_RAW_8215 { ExternalWritable := 'False'} : "UT00801_St_ConstAiRawData";   // AI Thermal Resistance - 3-wire (Pt10 climate - 3902)
      AI_RAW_8515 { ExternalWritable := 'False'} : "UT00801_St_ConstAiRawData";   // AI Thermal Resistance - 3-wire (Pt10 climate - 391)
      AI_RAW_8115 { ExternalWritable := 'False'} : "UT00801_St_ConstAiRawData";   // AI Thermal Resistance - 3-wire (Pt10 climate - 3916)
      AI_RAW_8315 { ExternalWritable := 'False'} : "UT00801_St_ConstAiRawData";   // AI Thermal Resistance - 3-wire (Pt10 climate - 392)
      AI_RAW_8014 { ExternalWritable := 'False'} : "UT00801_St_ConstAiRawData";   // AI Thermal Resistance - 3-wire (Pt10 standard - 3851)
      AI_RAW_8214 { ExternalWritable := 'False'} : "UT00801_St_ConstAiRawData";   // AI Thermal Resistance - 3-wire (Pt10 standard - 3902)
      AI_RAW_8514 { ExternalWritable := 'False'} : "UT00801_St_ConstAiRawData";   // AI Thermal Resistance - 3-wire (Pt10 standard - 391)
      AI_RAW_8114 { ExternalWritable := 'False'} : "UT00801_St_ConstAiRawData";   // AI Thermal Resistance - 3-wire (Pt10 standard - 3916)
      AI_RAW_8314 { ExternalWritable := 'False'} : "UT00801_St_ConstAiRawData";   // AI Thermal Resistance - 3-wire (Pt10 standard - 392)
      AI_RAW_8017 { ExternalWritable := 'False'} : "UT00801_St_ConstAiRawData";   // AI Thermal Resistance - 3-wire (Pt50 climate - 3851)
      AI_RAW_8217 { ExternalWritable := 'False'} : "UT00801_St_ConstAiRawData";   // AI Thermal Resistance - 3-wire (Pt50 climate - 3902)
      AI_RAW_8517 { ExternalWritable := 'False'} : "UT00801_St_ConstAiRawData";   // AI Thermal Resistance - 3-wire (Pt50 climate - 391)
      AI_RAW_8117 { ExternalWritable := 'False'} : "UT00801_St_ConstAiRawData";   // AI Thermal Resistance - 3-wire (Pt50 climate - 3916)
      AI_RAW_8317 { ExternalWritable := 'False'} : "UT00801_St_ConstAiRawData";   // AI Thermal Resistance - 3-wire (Pt50 climate - 392)
      AI_RAW_8016 { ExternalWritable := 'False'} : "UT00801_St_ConstAiRawData";   // AI Thermal Resistance - 3-wire (Pt50 standard - 3851)
      AI_RAW_8216 { ExternalWritable := 'False'} : "UT00801_St_ConstAiRawData";   // AI Thermal Resistance - 3-wire (Pt50 standard - 3902)
      AI_RAW_8516 { ExternalWritable := 'False'} : "UT00801_St_ConstAiRawData";   // AI Thermal Resistance - 3-wire (Pt50 standard - 391)
      AI_RAW_8116 { ExternalWritable := 'False'} : "UT00801_St_ConstAiRawData";   // AI Thermal Resistance - 3-wire (Pt50 standard - 3916)
      AI_RAW_8316 { ExternalWritable := 'False'} : "UT00801_St_ConstAiRawData";   // AI Thermal Resistance - 3-wire (Pt50 standard - 392)
      AI_RAW_8000 { ExternalWritable := 'False'} : "UT00801_St_ConstAiRawData";   // AI Thermal Resistance - 3-wire (Pt100 climate - 3851)
      AI_RAW_8200 { ExternalWritable := 'False'} : "UT00801_St_ConstAiRawData";   // AI Thermal Resistance - 3-wire (Pt100 climate - 3902)
      AI_RAW_8500 { ExternalWritable := 'False'} : "UT00801_St_ConstAiRawData";   // AI Thermal Resistance - 3-wire (Pt100 climate - 391)
      AI_RAW_8100 { ExternalWritable := 'False'} : "UT00801_St_ConstAiRawData";   // AI Thermal Resistance - 3-wire (Pt100 climate - 3916)
      AI_RAW_8300 { ExternalWritable := 'False'; S7_SetPoint := 'True'} : "UT00801_St_ConstAiRawData";   // AI Thermal Resistance - 3-wire (Pt100 climate - 392)
      AI_RAW_8002 { ExternalWritable := 'False'} : "UT00801_St_ConstAiRawData";   // AI Thermal Resistance - 3-wire (Pt100 standard - 3851)
   END_VAR
   VAR RETAIN
      AI_RAW_8202 { ExternalWritable := 'False'} : "UT00801_St_ConstAiRawData";   // AI Thermal Resistance - 3-wire (Pt100 standard - 3902)
   END_VAR
   VAR
      AI_RAW_8502 { ExternalWritable := 'False'} : "UT00801_St_ConstAiRawData";   // AI Thermal Resistance - 3-wire (Pt100 standard - 391)
      AI_RAW_8102 { ExternalWritable := 'False'} : "UT00801_St_ConstAiRawData";   // AI Thermal Resistance - 3-wire (Pt100 standard - 3916)
      AI_RAW_8302 { ExternalWritable := 'False'} : "UT00801_St_ConstAiRawData";   // AI Thermal Resistance - 3-wire (Pt100 standard - 392)
      AI_RAW_8007 { ExternalWritable := 'False'} : "UT00801_St_ConstAiRawData";   // AI Thermal Resistance - 3-wire (Pt200 climate - 3851)
      AI_RAW_8207 { ExternalWritable := 'False'} : "UT00801_St_ConstAiRawData";   // AI Thermal Resistance - 3-wire (Pt200 climate - 3902)
      AI_RAW_8507 { ExternalWritable := 'False'} : "UT00801_St_ConstAiRawData";   // AI Thermal Resistance - 3-wire (Pt200 climate - 391)
      AI_RAW_8107 { ExternalWritable := 'False'} : "UT00801_St_ConstAiRawData";   // AI Thermal Resistance - 3-wire (Pt200 climate - 3916)
      AI_RAW_8307 { ExternalWritable := 'False'} : "UT00801_St_ConstAiRawData";   // AI Thermal Resistance - 3-wire (Pt200 climate - 392)
      AI_RAW_800B { ExternalWritable := 'False'} : "UT00801_St_ConstAiRawData";   // AI Thermal Resistance - 3-wire (Pt200 standard - 3851)
      AI_RAW_820B { ExternalWritable := 'False'} : "UT00801_St_ConstAiRawData";   // AI Thermal Resistance - 3-wire (Pt200 standard - 3902)
      AI_RAW_850B { ExternalWritable := 'False'} : "UT00801_St_ConstAiRawData";   // AI Thermal Resistance - 3-wire (Pt200 standard - 391)
      AI_RAW_810B { ExternalWritable := 'False'} : "UT00801_St_ConstAiRawData";   // AI Thermal Resistance - 3-wire (Pt200 standard - 3916)
      AI_RAW_830B { ExternalWritable := 'False'} : "UT00801_St_ConstAiRawData";   // AI Thermal Resistance - 3-wire (Pt200 standard - 392)
      AI_RAW_8008 { ExternalWritable := 'False'} : "UT00801_St_ConstAiRawData";   // AI Thermal Resistance - 3-wire (Pt500 climate - 3851)
      AI_RAW_8208 { ExternalWritable := 'False'} : "UT00801_St_ConstAiRawData";   // AI Thermal Resistance - 3-wire (Pt500 climate - 3902)
      AI_RAW_8508 { ExternalWritable := 'False'} : "UT00801_St_ConstAiRawData";   // AI Thermal Resistance - 3-wire (Pt500 climate - 391)
      AI_RAW_8108 { ExternalWritable := 'False'} : "UT00801_St_ConstAiRawData";   // AI Thermal Resistance - 3-wire (Pt500 climate - 3916)
      AI_RAW_8308 { ExternalWritable := 'False'} : "UT00801_St_ConstAiRawData";   // AI Thermal Resistance - 3-wire (Pt500 climate - 392)
      AI_RAW_8004 { ExternalWritable := 'False'} : "UT00801_St_ConstAiRawData";   // AI Thermal Resistance - 3-wire (Pt500 standard - 3851)
      AI_RAW_8204 { ExternalWritable := 'False'} : "UT00801_St_ConstAiRawData";   // AI Thermal Resistance - 3-wire (Pt500 standard - 3902)
      AI_RAW_8504 { ExternalWritable := 'False'} : "UT00801_St_ConstAiRawData";   // AI Thermal Resistance - 3-wire (Pt500 standard - 391)
      AI_RAW_8104 { ExternalWritable := 'False'} : "UT00801_St_ConstAiRawData";   // AI Thermal Resistance - 3-wire (Pt500 standard - 3916)
      AI_RAW_8304 { ExternalWritable := 'False'} : "UT00801_St_ConstAiRawData";   // AI Thermal Resistance - 3-wire (Pt500 standard - 392)
      AI_RAW_8009 { ExternalWritable := 'False'} : "UT00801_St_ConstAiRawData";   // AI Thermal Resistance - 3-wire (Pt1000 climate - 3851)
      AI_RAW_8209 { ExternalWritable := 'False'} : "UT00801_St_ConstAiRawData";   // AI Thermal Resistance - 3-wire (Pt1000 climate - 3902)
      AI_RAW_8509 { ExternalWritable := 'False'} : "UT00801_St_ConstAiRawData";   // AI Thermal Resistance - 3-wire (Pt1000 climate - 391)
      AI_RAW_8109 { ExternalWritable := 'False'} : "UT00801_St_ConstAiRawData";   // AI Thermal Resistance - 3-wire (Pt1000 climate - 3916)
      AI_RAW_8309 { ExternalWritable := 'False'} : "UT00801_St_ConstAiRawData";   // AI Thermal Resistance - 3-wire (Pt1000 climate - 392)
      AI_RAW_8005 { ExternalWritable := 'False'} : "UT00801_St_ConstAiRawData";   // AI Thermal Resistance - 3-wire (Pt1000 standard - 3851)
      AI_RAW_8205 { ExternalWritable := 'False'} : "UT00801_St_ConstAiRawData";   // AI Thermal Resistance - 3-wire (Pt1000 standard - 3902)
      AI_RAW_8505 { ExternalWritable := 'False'} : "UT00801_St_ConstAiRawData";   // AI Thermal Resistance - 3-wire (Pt1000 standard - 391)
      AI_RAW_8105 { ExternalWritable := 'False'} : "UT00801_St_ConstAiRawData";   // AI Thermal Resistance - 3-wire (Pt1000 standard - 3916)
      AI_RAW_8305 { ExternalWritable := 'False'} : "UT00801_St_ConstAiRawData";   // AI Thermal Resistance - 3-wire (Pt1000 standard - 392)
      __________0160_0 { ExternalAccessible := 'False'; ExternalVisible := 'False'; ExternalWritable := 'False'} : Bool := false;
      __________0160_1 { ExternalAccessible := 'False'; ExternalVisible := 'False'; ExternalWritable := 'False'} : Bool := false;   // ▀▀▀▀ ANALOG INPUT SIGNAL — THERMOCOUPLE
      AI_RAW_A000 { ExternalWritable := 'False'} : "UT00801_St_ConstAiRawData";   // AI Thermocouple (Type B)
      AI_RAW_A00A { ExternalWritable := 'False'} : "UT00801_St_ConstAiRawData";   // AI Thermocouple (Type C)
      AI_RAW_A002 { ExternalWritable := 'False'} : "UT00801_St_ConstAiRawData";   // AI Thermocouple (Type E)
      AI_RAW_A005 { ExternalWritable := 'False'} : "UT00801_St_ConstAiRawData";   // AI Thermocouple (Type J)
      AI_RAW_A008 { ExternalWritable := 'False'} : "UT00801_St_ConstAiRawData";   // AI Thermocouple (Type K)
      AI_RAW_A001 { ExternalWritable := 'False'} : "UT00801_St_ConstAiRawData";   // AI Thermocouple (Type N)
      AI_RAW_A003 { ExternalWritable := 'False'} : "UT00801_St_ConstAiRawData";   // AI Thermocouple (Type R)
      AI_RAW_A004 { ExternalWritable := 'False'} : "UT00801_St_ConstAiRawData";   // AI Thermocouple (Type S)
      AI_RAW_A007 { ExternalWritable := 'False'} : "UT00801_St_ConstAiRawData";   // AI Thermocouple (Type T)
      AI_RAW_A00B { ExternalWritable := 'False'} : "UT00801_St_ConstAiRawData";   // AI Thermocouple (Type TXK/XCL)
   END_VAR
BEGIN
   // _DB_Header[0] : ▄▄▄▄▄▄▄▄▄▄▄▄▄▄▄▄▄▄▄▄▄▄▄▄▄▄▄▄▄▄▄▄ ＣＯＮＳＴＡＮＴＳ ▄▄
   // _DB_Header[2] : TITLE: SYSTEM CONSTANTS — ANALOG INPUT CARD TYPE, RANGE AND COEFFICIENTS
   // _DB_Header[4] : ▀▀▀▀▀▀▀▀▀▀▀▀▀▀▀▀▀▀▀▀▀▀▀▀▀▀▀▀▀▀▀▀▀▀▀▀▀▀▀▀▀▀▀▀
   // _DB_Header[5] : TYPE: STATIC
   // _DB_Header[6] : ▄▄▄▄▄▄▄▄▄▄▄▄▄▄▄▄▄▄▄▄▄▄▄▄▄▄▄▄▄▄▄▄▄▄▄▄▄▄▄▄ ʷᴵᴰ⁻ᵈʰᵐ ▄
   // _DB_Header[8] : DB00801_St_ConstAiRawData is a static data block that holds a full set of range, parameter and
   // _DB_Header[9] : descriptive data for all types of analog input card channels.
   // _DB_Header[11] : Each dataset is stored in a structure of user data type: UT00801_St_ConstAiRawData.
   // _DB_Header[12] : This structure is configured to hold all the data required by the card itself, any module accessing
   // _DB_Header[13] : an analog input and any supervisory system that is to display the type and configuration of the
   // _DB_Header[14] : input channel.
   // _DB_Header[16] : All the channel data is stored as constants and is used by all modules that have an interface
   // _DB_Header[17] : to an analog input card.
   // _DB_Header[19] : The purpose of the user data type and associated data block is to provide a consistent and
   // _DB_Header[20] : tested set of range, parameter and descriptive data that can be used directly by modules that
   // _DB_Header[21] : interface with analog input cards.
   // _DB_Header[23] : The ranges correspond to the numerical values returned by the card for a given type of analog
   // _DB_Header[24] : card signal. For example, a 4-20 mA card returns a numerical value of 0 at 4 mA ranging up to a
   // _DB_Header[25] : value of 27648 at 20 mA. The data specified in the UT00801 variable would have a lower limit of
   // _DB_Header[26] : 0 and an upper limit of 27648.
   // _DB_Header[28] : In addition, each dataset contains the parametric data that defines the particular channel type
   // _DB_Header[29] : and can be used to set a particular analog input channel to a particular type and range during
   // _DB_Header[30] : runtime. Each dataset also contains a textual description of the channel type,:
   // _DB_Header[31] : e.g. Current – 4 wire (4 mA to 20 mA)
   // _DB_Header[32] : for display and information purposes.
   // _DB_Header[34] : Finally, data associated with thermal resistance channel types also contain the real number
   // _DB_Header[35] : value of the spe-cific temperature coefficient that is to be applied to the channel.
   // _DB_Header[37] : The PDF version of the SMDS for this module is available online here:
   // _DB_Header[38] : http://psop.uk/pal-smds-db00801-p
   // _DB_Header[40] : ━━━ ⬙⬙⬙⬙⬙⬙ ━━━
   // _DB_Header[42] : ▄▄▄▄▄▄▄▄▄▄▄▄▄▄▄▄▄▄▄▄▄▄▄▄▄▄▄▄▄▄▄▄▄▄▄▄▄▄▄▄▄▄▄▄
   // _DB_Header[43] : MODIFICATION HISTORY
   // _DB_Header[45] : This is a summary of the recent software modifications made to this block (most recent at top)
   // _DB_Header[47] : ―――――――――――――――――――――――――――――――――――――――――――
   // _DB_Header[48] : DATE REVISION MASTER BRANCH DEV
   // _DB_Header[49] : (nnn.amm) COMMIT TAG (Base ---> Merge) BRANCH Author
   // _DB_Header[50] : ———————————————————————————————————————————
   // _DB_Header[51] : 2024.05.15 001.000 D0017A-000.104 D0017 N/A D0017A M. Gledhill
   // _DB_Header[52] : DB00801 — RELEASED FOR USE
   // _DB_Header[54] : 2024.05.03 000.801 D0017A-000.102 D0017 N/A D0017A M. Gledhill
   // _DB_Header[55] : DB00801 Block populated
   // _DB_Header[56] : 2024.04.09 000.101 D0017A-000.101 D0017 N/A D0017A M. Gledhill
   // _DB_Header[57] : DB00801 Block created
   // _DB_Header[58] : ———————————————————————————————————————————
   // _DB_Header[59] : Where: nnn = Major revision
   // _DB_Header[60] : a = Type (1-7 Development, 8 Proving, 9 Qualification, 0 Release)
   // _DB_Header[61] : mm = Minor revision (must be 00 if a = 0)
   // _DB_Header[62] : Block properties version number should be set to nn.a (only one decimal place)
   // _DB_Header[64] : ██████████████ █ █ █ █ END █ █ █ █ ██████████████
   revInfo.REV_BLOCK := 'DB00801';
   revInfo.REV_NUMBER := '001.000';
   revInfo.REV_DATE := '2024-05-15';
   revInfo.REV_AUTHOR := 'M. Gledhill';
   AI_RAW_0000.revInfo.REV_BLOCK := 'UT00801';
   AI_RAW_0000.revInfo.REV_NUMBER := '001.000';
   AI_RAW_0000.revInfo.REV_DATE := '2024-04-09';
   AI_RAW_0000.revInfo.REV_AUTHOR := 'M. Gledhill';
   AI_RAW_0000.___________0010_0 := false;
   AI_RAW_0000.___________0010_1 := false;
   AI_RAW_0000.AI_CODE := 16#0000;
   AI_RAW_0000.___________0020_0 := false;
   AI_RAW_0000.___________0020_1 := false;
   AI_RAW_0000.RAW_MIN := 0;
   AI_RAW_0000.RAW_MAX := 0;
   AI_RAW_0000.RAW_DESC := 'User defined signal type';
   AI_RAW_0000.___________0030_1 := false;
   AI_RAW_0000.___________0030_2 := false;
   AI_RAW_0000.PARAM_TYPE := 16#00;
   AI_RAW_0000.PARAM_RANGE := 16#00;
   AI_RAW_0000.PARAM_COEF := 16#00;
   AI_RAW_0000.___________0040_1 := false;
   AI_RAW_0000.___________0040_2 := false;
   AI_RAW_0000.VALUE_COEF := 0.0;
   AI_RAW_1000.revInfo.REV_BLOCK := 'UT00801';
   AI_RAW_1000.revInfo.REV_NUMBER := '001.000';
   AI_RAW_1000.revInfo.REV_DATE := '2024-04-09';
   AI_RAW_1000.revInfo.REV_AUTHOR := 'M. Gledhill';
   AI_RAW_1000.___________0010_0 := false;
   AI_RAW_1000.___________0010_1 := false;
   AI_RAW_1000.AI_CODE := 16#1000;
   AI_RAW_1000.___________0020_0 := false;
   AI_RAW_1000.___________0020_1 := false;
   AI_RAW_1000.RAW_MIN := -27648;
   AI_RAW_1000.RAW_MAX := 27648;
   AI_RAW_1000.RAW_DESC := 'Voltage (-25 mV to +25 mV)';
   AI_RAW_1000.___________0030_1 := false;
   AI_RAW_1000.___________0030_2 := false;
   AI_RAW_1000.PARAM_TYPE := 16#01;
   AI_RAW_1000.PARAM_RANGE := 16#00;
   AI_RAW_1000.PARAM_COEF := 16#00;
   AI_RAW_1000.___________0040_1 := false;
   AI_RAW_1000.___________0040_2 := false;
   AI_RAW_1000.VALUE_COEF := 0.0;
   AI_RAW_1001.revInfo.REV_BLOCK := 'UT00801';
   AI_RAW_1001.revInfo.REV_NUMBER := '001.000';
   AI_RAW_1001.revInfo.REV_DATE := '2024-04-09';
   AI_RAW_1001.revInfo.REV_AUTHOR := 'M. Gledhill';
   AI_RAW_1001.___________0010_0 := false;
   AI_RAW_1001.___________0010_1 := false;
   AI_RAW_1001.AI_CODE := 16#1001;
   AI_RAW_1001.___________0020_0 := false;
   AI_RAW_1001.___________0020_1 := false;
   AI_RAW_1001.RAW_MIN := -27648;
   AI_RAW_1001.RAW_MAX := 27648;
   AI_RAW_1001.RAW_DESC := 'Voltage (-50 mV to +50 mV)';
   AI_RAW_1001.___________0030_1 := false;
   AI_RAW_1001.___________0030_2 := false;
   AI_RAW_1001.PARAM_TYPE := 16#01;
   AI_RAW_1001.PARAM_RANGE := 16#01;
   AI_RAW_1001.PARAM_COEF := 16#00;
   AI_RAW_1001.___________0040_1 := false;
   AI_RAW_1001.___________0040_2 := false;
   AI_RAW_1001.VALUE_COEF := 0.0;
   AI_RAW_1002.revInfo.REV_BLOCK := 'UT00801';
   AI_RAW_1002.revInfo.REV_NUMBER := '001.000';
   AI_RAW_1002.revInfo.REV_DATE := '2024-04-09';
   AI_RAW_1002.revInfo.REV_AUTHOR := 'M. Gledhill';
   AI_RAW_1002.___________0010_0 := false;
   AI_RAW_1002.___________0010_1 := false;
   AI_RAW_1002.AI_CODE := 16#1002;
   AI_RAW_1002.___________0020_0 := false;
   AI_RAW_1002.___________0020_1 := false;
   AI_RAW_1002.RAW_MIN := -27648;
   AI_RAW_1002.RAW_MAX := 27648;
   AI_RAW_1002.RAW_DESC := 'Voltage (-80 mV to +80 mV)';
   AI_RAW_1002.___________0030_1 := false;
   AI_RAW_1002.___________0030_2 := false;
   AI_RAW_1002.PARAM_TYPE := 16#01;
   AI_RAW_1002.PARAM_RANGE := 16#02;
   AI_RAW_1002.PARAM_COEF := 16#00;
   AI_RAW_1002.___________0040_1 := false;
   AI_RAW_1002.___________0040_2 := false;
   AI_RAW_1002.VALUE_COEF := 0.0;
   AI_RAW_1003.revInfo.REV_BLOCK := 'UT00801';
   AI_RAW_1003.revInfo.REV_NUMBER := '001.000';
   AI_RAW_1003.revInfo.REV_DATE := '2024-04-09';
   AI_RAW_1003.revInfo.REV_AUTHOR := 'M. Gledhill';
   AI_RAW_1003.___________0010_0 := false;
   AI_RAW_1003.___________0010_1 := false;
   AI_RAW_1003.AI_CODE := 16#1003;
   AI_RAW_1003.___________0020_0 := false;
   AI_RAW_1003.___________0020_1 := false;
   AI_RAW_1003.RAW_MIN := -27648;
   AI_RAW_1003.RAW_MAX := 27648;
   AI_RAW_1003.RAW_DESC := 'Voltage (-250 mV to +250 mV)';
   AI_RAW_1003.___________0030_1 := false;
   AI_RAW_1003.___________0030_2 := false;
   AI_RAW_1003.PARAM_TYPE := 16#01;
   AI_RAW_1003.PARAM_RANGE := 16#03;
   AI_RAW_1003.PARAM_COEF := 16#00;
   AI_RAW_1003.___________0040_1 := false;
   AI_RAW_1003.___________0040_2 := false;
   AI_RAW_1003.VALUE_COEF := 0.0;
   AI_RAW_1004.revInfo.REV_BLOCK := 'UT00801';
   AI_RAW_1004.revInfo.REV_NUMBER := '001.000';
   AI_RAW_1004.revInfo.REV_DATE := '2024-04-09';
   AI_RAW_1004.revInfo.REV_AUTHOR := 'M. Gledhill';
   AI_RAW_1004.___________0010_0 := false;
   AI_RAW_1004.___________0010_1 := false;
   AI_RAW_1004.AI_CODE := 16#1004;
   AI_RAW_1004.___________0020_0 := false;
   AI_RAW_1004.___________0020_1 := false;
   AI_RAW_1004.RAW_MIN := -27648;
   AI_RAW_1004.RAW_MAX := 27648;
   AI_RAW_1004.RAW_DESC := 'Voltage (-500 mV to +500 mV)';
   AI_RAW_1004.___________0030_1 := false;
   AI_RAW_1004.___________0030_2 := false;
   AI_RAW_1004.PARAM_TYPE := 16#01;
   AI_RAW_1004.PARAM_RANGE := 16#04;
   AI_RAW_1004.PARAM_COEF := 16#00;
   AI_RAW_1004.___________0040_1 := false;
   AI_RAW_1004.___________0040_2 := false;
   AI_RAW_1004.VALUE_COEF := 0.0;
   AI_RAW_1005.revInfo.REV_BLOCK := 'UT00801';
   AI_RAW_1005.revInfo.REV_NUMBER := '001.000';
   AI_RAW_1005.revInfo.REV_DATE := '2024-04-09';
   AI_RAW_1005.revInfo.REV_AUTHOR := 'M. Gledhill';
   AI_RAW_1005.___________0010_0 := false;
   AI_RAW_1005.___________0010_1 := false;
   AI_RAW_1005.AI_CODE := 16#1005;
   AI_RAW_1005.___________0020_0 := false;
   AI_RAW_1005.___________0020_1 := false;
   AI_RAW_1005.RAW_MIN := -27648;
   AI_RAW_1005.RAW_MAX := 27648;
   AI_RAW_1005.RAW_DESC := 'Voltage (-1 V to +1 V)';
   AI_RAW_1005.___________0030_1 := false;
   AI_RAW_1005.___________0030_2 := false;
   AI_RAW_1005.PARAM_TYPE := 16#01;
   AI_RAW_1005.PARAM_RANGE := 16#05;
   AI_RAW_1005.PARAM_COEF := 16#00;
   AI_RAW_1005.___________0040_1 := false;
   AI_RAW_1005.___________0040_2 := false;
   AI_RAW_1005.VALUE_COEF := 0.0;
   AI_RAW_1007.revInfo.REV_BLOCK := 'UT00801';
   AI_RAW_1007.revInfo.REV_NUMBER := '001.000';
   AI_RAW_1007.revInfo.REV_DATE := '2024-04-09';
   AI_RAW_1007.revInfo.REV_AUTHOR := 'M. Gledhill';
   AI_RAW_1007.___________0010_0 := false;
   AI_RAW_1007.___________0010_1 := false;
   AI_RAW_1007.AI_CODE := 16#1007;
   AI_RAW_1007.___________0020_0 := false;
   AI_RAW_1007.___________0020_1 := false;
   AI_RAW_1007.RAW_MIN := -27648;
   AI_RAW_1007.RAW_MAX := 27648;
   AI_RAW_1007.RAW_DESC := 'Voltage (-2.5 V to +2.5 V)';
   AI_RAW_1007.___________0030_1 := false;
   AI_RAW_1007.___________0030_2 := false;
   AI_RAW_1007.PARAM_TYPE := 16#01;
   AI_RAW_1007.PARAM_RANGE := 16#07;
   AI_RAW_1007.PARAM_COEF := 16#00;
   AI_RAW_1007.___________0040_1 := false;
   AI_RAW_1007.___________0040_2 := false;
   AI_RAW_1007.VALUE_COEF := 0.0;
   AI_RAW_1008.revInfo.REV_BLOCK := 'UT00801';
   AI_RAW_1008.revInfo.REV_NUMBER := '001.000';
   AI_RAW_1008.revInfo.REV_DATE := '2024-04-09';
   AI_RAW_1008.revInfo.REV_AUTHOR := 'M. Gledhill';
   AI_RAW_1008.___________0010_0 := false;
   AI_RAW_1008.___________0010_1 := false;
   AI_RAW_1008.AI_CODE := 16#1008;
   AI_RAW_1008.___________0020_0 := false;
   AI_RAW_1008.___________0020_1 := false;
   AI_RAW_1008.RAW_MIN := -27648;
   AI_RAW_1008.RAW_MAX := 27648;
   AI_RAW_1008.RAW_DESC := 'Voltage (-5 V to +5 V)';
   AI_RAW_1008.___________0030_1 := false;
   AI_RAW_1008.___________0030_2 := false;
   AI_RAW_1008.PARAM_TYPE := 16#01;
   AI_RAW_1008.PARAM_RANGE := 16#08;
   AI_RAW_1008.PARAM_COEF := 16#00;
   AI_RAW_1008.___________0040_1 := false;
   AI_RAW_1008.___________0040_2 := false;
   AI_RAW_1008.VALUE_COEF := 0.0;
   AI_RAW_1009.revInfo.REV_BLOCK := 'UT00801';
   AI_RAW_1009.revInfo.REV_NUMBER := '001.000';
   AI_RAW_1009.revInfo.REV_DATE := '2024-04-09';
   AI_RAW_1009.revInfo.REV_AUTHOR := 'M. Gledhill';
   AI_RAW_1009.___________0010_0 := false;
   AI_RAW_1009.___________0010_1 := false;
   AI_RAW_1009.AI_CODE := 16#1009;
   AI_RAW_1009.___________0020_0 := false;
   AI_RAW_1009.___________0020_1 := false;
   AI_RAW_1009.RAW_MIN := -27648;
   AI_RAW_1009.RAW_MAX := 27648;
   AI_RAW_1009.RAW_DESC := 'Voltage (-10 V to +10 V)';
   AI_RAW_1009.___________0030_1 := false;
   AI_RAW_1009.___________0030_2 := false;
   AI_RAW_1009.PARAM_TYPE := 16#01;
   AI_RAW_1009.PARAM_RANGE := 16#09;
   AI_RAW_1009.PARAM_COEF := 16#00;
   AI_RAW_1009.___________0040_1 := false;
   AI_RAW_1009.___________0040_2 := false;
   AI_RAW_1009.VALUE_COEF := 0.0;
   AI_RAW_100A.revInfo.REV_BLOCK := 'UT00801';
   AI_RAW_100A.revInfo.REV_NUMBER := '001.000';
   AI_RAW_100A.revInfo.REV_DATE := '2024-04-09';
   AI_RAW_100A.revInfo.REV_AUTHOR := 'M. Gledhill';
   AI_RAW_100A.___________0010_0 := false;
   AI_RAW_100A.___________0010_1 := false;
   AI_RAW_100A.AI_CODE := 16#100A;
   AI_RAW_100A.___________0020_0 := false;
   AI_RAW_100A.___________0020_1 := false;
   AI_RAW_100A.RAW_MIN := 0;
   AI_RAW_100A.RAW_MAX := 27648;
   AI_RAW_100A.RAW_DESC := 'Voltage (1 V to 5 V)';
   AI_RAW_100A.___________0030_1 := false;
   AI_RAW_100A.___________0030_2 := false;
   AI_RAW_100A.PARAM_TYPE := 16#01;
   AI_RAW_100A.PARAM_RANGE := 16#0A;
   AI_RAW_100A.PARAM_COEF := 16#00;
   AI_RAW_100A.___________0040_1 := false;
   AI_RAW_100A.___________0040_2 := false;
   AI_RAW_100A.VALUE_COEF := 0.0;
   AI_RAW_2002.revInfo.REV_BLOCK := 'UT00801';
   AI_RAW_2002.revInfo.REV_NUMBER := '001.000';
   AI_RAW_2002.revInfo.REV_DATE := '2024-04-09';
   AI_RAW_2002.revInfo.REV_AUTHOR := 'M. Gledhill';
   AI_RAW_2002.___________0010_0 := false;
   AI_RAW_2002.___________0010_1 := false;
   AI_RAW_2002.AI_CODE := 16#2002;
   AI_RAW_2002.___________0020_0 := false;
   AI_RAW_2002.___________0020_1 := false;
   AI_RAW_2002.RAW_MIN := 0;
   AI_RAW_2002.RAW_MAX := 27648;
   AI_RAW_2002.RAW_DESC := 'Current - 4-wire (0 mA to 20 mA)';
   AI_RAW_2002.___________0030_1 := false;
   AI_RAW_2002.___________0030_2 := false;
   AI_RAW_2002.PARAM_TYPE := 16#02;
   AI_RAW_2002.PARAM_RANGE := 16#02;
   AI_RAW_2002.PARAM_COEF := 16#00;
   AI_RAW_2002.___________0040_1 := false;
   AI_RAW_2002.___________0040_2 := false;
   AI_RAW_2002.VALUE_COEF := 0.0;
   AI_RAW_2003.revInfo.REV_BLOCK := 'UT00801';
   AI_RAW_2003.revInfo.REV_NUMBER := '001.000';
   AI_RAW_2003.revInfo.REV_DATE := '2024-04-09';
   AI_RAW_2003.revInfo.REV_AUTHOR := 'M. Gledhill';
   AI_RAW_2003.___________0010_0 := false;
   AI_RAW_2003.___________0010_1 := false;
   AI_RAW_2003.AI_CODE := 16#2003;
   AI_RAW_2003.___________0020_0 := false;
   AI_RAW_2003.___________0020_1 := false;
   AI_RAW_2003.RAW_MIN := 0;
   AI_RAW_2003.RAW_MAX := 27648;
   AI_RAW_2003.RAW_DESC := 'Current - 4-wire (4 mA to 20 mA)';
   AI_RAW_2003.___________0030_1 := false;
   AI_RAW_2003.___________0030_2 := false;
   AI_RAW_2003.PARAM_TYPE := 16#02;
   AI_RAW_2003.PARAM_RANGE := 16#03;
   AI_RAW_2003.PARAM_COEF := 16#00;
   AI_RAW_2003.___________0040_1 := false;
   AI_RAW_2003.___________0040_2 := false;
   AI_RAW_2003.VALUE_COEF := 0.0;
   AI_RAW_2004.revInfo.REV_BLOCK := 'UT00801';
   AI_RAW_2004.revInfo.REV_NUMBER := '001.000';
   AI_RAW_2004.revInfo.REV_DATE := '2024-04-09';
   AI_RAW_2004.revInfo.REV_AUTHOR := 'M. Gledhill';
   AI_RAW_2004.___________0010_0 := false;
   AI_RAW_2004.___________0010_1 := false;
   AI_RAW_2004.AI_CODE := 16#2004;
   AI_RAW_2004.___________0020_0 := false;
   AI_RAW_2004.___________0020_1 := false;
   AI_RAW_2004.RAW_MIN := -27648;
   AI_RAW_2004.RAW_MAX := 27648;
   AI_RAW_2004.RAW_DESC := 'Current - 4-wire (-20 mA to +20 mA)';
   AI_RAW_2004.___________0030_1 := false;
   AI_RAW_2004.___________0030_2 := false;
   AI_RAW_2004.PARAM_TYPE := 16#02;
   AI_RAW_2004.PARAM_RANGE := 16#04;
   AI_RAW_2004.PARAM_COEF := 16#00;
   AI_RAW_2004.___________0040_1 := false;
   AI_RAW_2004.___________0040_2 := false;
   AI_RAW_2004.VALUE_COEF := 0.0;
   AI_RAW_3003.revInfo.REV_BLOCK := 'UT00801';
   AI_RAW_3003.revInfo.REV_NUMBER := '001.000';
   AI_RAW_3003.revInfo.REV_DATE := '2024-04-09';
   AI_RAW_3003.revInfo.REV_AUTHOR := 'M. Gledhill';
   AI_RAW_3003.___________0010_0 := false;
   AI_RAW_3003.___________0010_1 := false;
   AI_RAW_3003.AI_CODE := 16#3003;
   AI_RAW_3003.___________0020_0 := false;
   AI_RAW_3003.___________0020_1 := false;
   AI_RAW_3003.RAW_MIN := 0;
   AI_RAW_3003.RAW_MAX := 27648;
   AI_RAW_3003.RAW_DESC := 'Current - 2-wire (4 mA to 20 mA)';
   AI_RAW_3003.___________0030_1 := false;
   AI_RAW_3003.___________0030_2 := false;
   AI_RAW_3003.PARAM_TYPE := 16#03;
   AI_RAW_3003.PARAM_RANGE := 16#03;
   AI_RAW_3003.PARAM_COEF := 16#00;
   AI_RAW_3003.___________0040_1 := false;
   AI_RAW_3003.___________0040_2 := false;
   AI_RAW_3003.VALUE_COEF := 0.0;
   AI_RAW_4001.revInfo.REV_BLOCK := 'UT00801';
   AI_RAW_4001.revInfo.REV_NUMBER := '001.000';
   AI_RAW_4001.revInfo.REV_DATE := '2024-04-09';
   AI_RAW_4001.revInfo.REV_AUTHOR := 'M. Gledhill';
   AI_RAW_4001.___________0010_0 := false;
   AI_RAW_4001.___________0010_1 := false;
   AI_RAW_4001.AI_CODE := 16#4001;
   AI_RAW_4001.___________0020_0 := false;
   AI_RAW_4001.___________0020_1 := false;
   AI_RAW_4001.RAW_MIN := 0;
   AI_RAW_4001.RAW_MAX := 27648;
   AI_RAW_4001.RAW_DESC := 'Resistance - 4-wire (150 Ohm)';
   AI_RAW_4001.___________0030_1 := false;
   AI_RAW_4001.___________0030_2 := false;
   AI_RAW_4001.PARAM_TYPE := 16#04;
   AI_RAW_4001.PARAM_RANGE := 16#01;
   AI_RAW_4001.PARAM_COEF := 16#00;
   AI_RAW_4001.___________0040_1 := false;
   AI_RAW_4001.___________0040_2 := false;
   AI_RAW_4001.VALUE_COEF := 0.0;
   AI_RAW_4002.revInfo.REV_BLOCK := 'UT00801';
   AI_RAW_4002.revInfo.REV_NUMBER := '001.000';
   AI_RAW_4002.revInfo.REV_DATE := '2024-04-09';
   AI_RAW_4002.revInfo.REV_AUTHOR := 'M. Gledhill';
   AI_RAW_4002.___________0010_0 := false;
   AI_RAW_4002.___________0010_1 := false;
   AI_RAW_4002.AI_CODE := 16#4002;
   AI_RAW_4002.___________0020_0 := false;
   AI_RAW_4002.___________0020_1 := false;
   AI_RAW_4002.RAW_MIN := 0;
   AI_RAW_4002.RAW_MAX := 27648;
   AI_RAW_4002.RAW_DESC := 'Resistance - 4-wire (300 Ohm)';
   AI_RAW_4002.___________0030_1 := false;
   AI_RAW_4002.___________0030_2 := false;
   AI_RAW_4002.PARAM_TYPE := 16#04;
   AI_RAW_4002.PARAM_RANGE := 16#02;
   AI_RAW_4002.PARAM_COEF := 16#00;
   AI_RAW_4002.___________0040_1 := false;
   AI_RAW_4002.___________0040_2 := false;
   AI_RAW_4002.VALUE_COEF := 0.0;
   AI_RAW_4003.revInfo.REV_BLOCK := 'UT00801';
   AI_RAW_4003.revInfo.REV_NUMBER := '001.000';
   AI_RAW_4003.revInfo.REV_DATE := '2024-04-09';
   AI_RAW_4003.revInfo.REV_AUTHOR := 'M. Gledhill';
   AI_RAW_4003.___________0010_0 := false;
   AI_RAW_4003.___________0010_1 := false;
   AI_RAW_4003.AI_CODE := 16#4003;
   AI_RAW_4003.___________0020_0 := false;
   AI_RAW_4003.___________0020_1 := false;
   AI_RAW_4003.RAW_MIN := 0;
   AI_RAW_4003.RAW_MAX := 27648;
   AI_RAW_4003.RAW_DESC := 'Resistance - 4-wire (600 Ohm)';
   AI_RAW_4003.___________0030_1 := false;
   AI_RAW_4003.___________0030_2 := false;
   AI_RAW_4003.PARAM_TYPE := 16#04;
   AI_RAW_4003.PARAM_RANGE := 16#03;
   AI_RAW_4003.PARAM_COEF := 16#00;
   AI_RAW_4003.___________0040_1 := false;
   AI_RAW_4003.___________0040_2 := false;
   AI_RAW_4003.VALUE_COEF := 0.0;
   AI_RAW_4005.revInfo.REV_BLOCK := 'UT00801';
   AI_RAW_4005.revInfo.REV_NUMBER := '001.000';
   AI_RAW_4005.revInfo.REV_DATE := '2024-04-09';
   AI_RAW_4005.revInfo.REV_AUTHOR := 'M. Gledhill';
   AI_RAW_4005.___________0010_0 := false;
   AI_RAW_4005.___________0010_1 := false;
   AI_RAW_4005.AI_CODE := 16#4005;
   AI_RAW_4005.___________0020_0 := false;
   AI_RAW_4005.___________0020_1 := false;
   AI_RAW_4005.RAW_MIN := 0;
   AI_RAW_4005.RAW_MAX := 27648;
   AI_RAW_4005.RAW_DESC := 'Resistance - 4-wire (6000 Ohm)';
   AI_RAW_4005.___________0030_1 := false;
   AI_RAW_4005.___________0030_2 := false;
   AI_RAW_4005.PARAM_TYPE := 16#04;
   AI_RAW_4005.PARAM_RANGE := 16#05;
   AI_RAW_4005.PARAM_COEF := 16#00;
   AI_RAW_4005.___________0040_1 := false;
   AI_RAW_4005.___________0040_2 := false;
   AI_RAW_4005.VALUE_COEF := 0.0;
   AI_RAW_5001.revInfo.REV_BLOCK := 'UT00801';
   AI_RAW_5001.revInfo.REV_NUMBER := '001.000';
   AI_RAW_5001.revInfo.REV_DATE := '2024-04-09';
   AI_RAW_5001.revInfo.REV_AUTHOR := 'M. Gledhill';
   AI_RAW_5001.___________0010_0 := false;
   AI_RAW_5001.___________0010_1 := false;
   AI_RAW_5001.AI_CODE := 16#5001;
   AI_RAW_5001.___________0020_0 := false;
   AI_RAW_5001.___________0020_1 := false;
   AI_RAW_5001.RAW_MIN := 0;
   AI_RAW_5001.RAW_MAX := 27648;
   AI_RAW_5001.RAW_DESC := 'Resistance - 3-wire (150 Ohm)';
   AI_RAW_5001.___________0030_1 := false;
   AI_RAW_5001.___________0030_2 := false;
   AI_RAW_5001.PARAM_TYPE := 16#05;
   AI_RAW_5001.PARAM_RANGE := 16#01;
   AI_RAW_5001.PARAM_COEF := 16#00;
   AI_RAW_5001.___________0040_1 := false;
   AI_RAW_5001.___________0040_2 := false;
   AI_RAW_5001.VALUE_COEF := 0.0;
   AI_RAW_5002.revInfo.REV_BLOCK := 'UT00801';
   AI_RAW_5002.revInfo.REV_NUMBER := '001.000';
   AI_RAW_5002.revInfo.REV_DATE := '2024-04-09';
   AI_RAW_5002.revInfo.REV_AUTHOR := 'M. Gledhill';
   AI_RAW_5002.___________0010_0 := false;
   AI_RAW_5002.___________0010_1 := false;
   AI_RAW_5002.AI_CODE := 16#5002;
   AI_RAW_5002.___________0020_0 := false;
   AI_RAW_5002.___________0020_1 := false;
   AI_RAW_5002.RAW_MIN := 0;
   AI_RAW_5002.RAW_MAX := 27648;
   AI_RAW_5002.RAW_DESC := 'Resistance - 3-wire (300 Ohm)';
   AI_RAW_5002.___________0030_1 := false;
   AI_RAW_5002.___________0030_2 := false;
   AI_RAW_5002.PARAM_TYPE := 16#05;
   AI_RAW_5002.PARAM_RANGE := 16#02;
   AI_RAW_5002.PARAM_COEF := 16#00;
   AI_RAW_5002.___________0040_1 := false;
   AI_RAW_5002.___________0040_2 := false;
   AI_RAW_5002.VALUE_COEF := 0.0;
   AI_RAW_5003.revInfo.REV_BLOCK := 'UT00801';
   AI_RAW_5003.revInfo.REV_NUMBER := '001.000';
   AI_RAW_5003.revInfo.REV_DATE := '2024-04-09';
   AI_RAW_5003.revInfo.REV_AUTHOR := 'M. Gledhill';
   AI_RAW_5003.___________0010_0 := false;
   AI_RAW_5003.___________0010_1 := false;
   AI_RAW_5003.AI_CODE := 16#5003;
   AI_RAW_5003.___________0020_0 := false;
   AI_RAW_5003.___________0020_1 := false;
   AI_RAW_5003.RAW_MIN := 0;
   AI_RAW_5003.RAW_MAX := 27648;
   AI_RAW_5003.RAW_DESC := 'Resistance - 3-wire (600 Ohm)';
   AI_RAW_5003.___________0030_1 := false;
   AI_RAW_5003.___________0030_2 := false;
   AI_RAW_5003.PARAM_TYPE := 16#05;
   AI_RAW_5003.PARAM_RANGE := 16#03;
   AI_RAW_5003.PARAM_COEF := 16#00;
   AI_RAW_5003.___________0040_1 := false;
   AI_RAW_5003.___________0040_2 := false;
   AI_RAW_5003.VALUE_COEF := 0.0;
   AI_RAW_5005.revInfo.REV_BLOCK := 'UT00801';
   AI_RAW_5005.revInfo.REV_NUMBER := '001.000';
   AI_RAW_5005.revInfo.REV_DATE := '2024-04-09';
   AI_RAW_5005.revInfo.REV_AUTHOR := 'M. Gledhill';
   AI_RAW_5005.___________0010_0 := false;
   AI_RAW_5005.___________0010_1 := false;
   AI_RAW_5005.AI_CODE := 16#5005;
   AI_RAW_5005.___________0020_0 := false;
   AI_RAW_5005.___________0020_1 := false;
   AI_RAW_5005.RAW_MIN := 0;
   AI_RAW_5005.RAW_MAX := 27648;
   AI_RAW_5005.RAW_DESC := 'Resistance - 3-wire (6000 Ohm)';
   AI_RAW_5005.___________0030_1 := false;
   AI_RAW_5005.___________0030_2 := false;
   AI_RAW_5005.PARAM_TYPE := 16#05;
   AI_RAW_5005.PARAM_RANGE := 16#05;
   AI_RAW_5005.PARAM_COEF := 16#00;
   AI_RAW_5005.___________0040_1 := false;
   AI_RAW_5005.___________0040_2 := false;
   AI_RAW_5005.VALUE_COEF := 0.0;
   AI_RAW_6001.revInfo.REV_BLOCK := 'UT00801';
   AI_RAW_6001.revInfo.REV_NUMBER := '001.000';
   AI_RAW_6001.revInfo.REV_DATE := '2024-04-09';
   AI_RAW_6001.revInfo.REV_AUTHOR := 'M. Gledhill';
   AI_RAW_6001.___________0010_0 := false;
   AI_RAW_6001.___________0010_1 := false;
   AI_RAW_6001.AI_CODE := 16#6001;
   AI_RAW_6001.___________0020_0 := false;
   AI_RAW_6001.___________0020_1 := false;
   AI_RAW_6001.RAW_MIN := 0;
   AI_RAW_6001.RAW_MAX := 27648;
   AI_RAW_6001.RAW_DESC := 'Resistance - 2-wire (150 Ohm)';
   AI_RAW_6001.___________0030_1 := false;
   AI_RAW_6001.___________0030_2 := false;
   AI_RAW_6001.PARAM_TYPE := 16#06;
   AI_RAW_6001.PARAM_RANGE := 16#01;
   AI_RAW_6001.PARAM_COEF := 16#00;
   AI_RAW_6001.___________0040_1 := false;
   AI_RAW_6001.___________0040_2 := false;
   AI_RAW_6001.VALUE_COEF := 0.0;
   AI_RAW_6002.revInfo.REV_BLOCK := 'UT00801';
   AI_RAW_6002.revInfo.REV_NUMBER := '001.000';
   AI_RAW_6002.revInfo.REV_DATE := '2024-04-09';
   AI_RAW_6002.revInfo.REV_AUTHOR := 'M. Gledhill';
   AI_RAW_6002.___________0010_0 := false;
   AI_RAW_6002.___________0010_1 := false;
   AI_RAW_6002.AI_CODE := 16#6002;
   AI_RAW_6002.___________0020_0 := false;
   AI_RAW_6002.___________0020_1 := false;
   AI_RAW_6002.RAW_MIN := 0;
   AI_RAW_6002.RAW_MAX := 27648;
   AI_RAW_6002.RAW_DESC := 'Resistance - 2-wire (300 Ohm)';
   AI_RAW_6002.___________0030_1 := false;
   AI_RAW_6002.___________0030_2 := false;
   AI_RAW_6002.PARAM_TYPE := 16#06;
   AI_RAW_6002.PARAM_RANGE := 16#02;
   AI_RAW_6002.PARAM_COEF := 16#00;
   AI_RAW_6002.___________0040_1 := false;
   AI_RAW_6002.___________0040_2 := false;
   AI_RAW_6002.VALUE_COEF := 0.0;
   AI_RAW_6003.revInfo.REV_BLOCK := 'UT00801';
   AI_RAW_6003.revInfo.REV_NUMBER := '001.000';
   AI_RAW_6003.revInfo.REV_DATE := '2024-04-09';
   AI_RAW_6003.revInfo.REV_AUTHOR := 'M. Gledhill';
   AI_RAW_6003.___________0010_0 := false;
   AI_RAW_6003.___________0010_1 := false;
   AI_RAW_6003.AI_CODE := 16#6003;
   AI_RAW_6003.___________0020_0 := false;
   AI_RAW_6003.___________0020_1 := false;
   AI_RAW_6003.RAW_MIN := 0;
   AI_RAW_6003.RAW_MAX := 27648;
   AI_RAW_6003.RAW_DESC := 'Resistance - 2-wire (600 Ohm)';
   AI_RAW_6003.___________0030_1 := false;
   AI_RAW_6003.___________0030_2 := false;
   AI_RAW_6003.PARAM_TYPE := 16#06;
   AI_RAW_6003.PARAM_RANGE := 16#03;
   AI_RAW_6003.PARAM_COEF := 16#00;
   AI_RAW_6003.___________0040_1 := false;
   AI_RAW_6003.___________0040_2 := false;
   AI_RAW_6003.VALUE_COEF := 0.0;
   AI_RAW_6005.revInfo.REV_BLOCK := 'UT00801';
   AI_RAW_6005.revInfo.REV_NUMBER := '001.000';
   AI_RAW_6005.revInfo.REV_DATE := '2024-04-09';
   AI_RAW_6005.revInfo.REV_AUTHOR := 'M. Gledhill';
   AI_RAW_6005.___________0010_0 := false;
   AI_RAW_6005.___________0010_1 := false;
   AI_RAW_6005.AI_CODE := 16#6005;
   AI_RAW_6005.___________0020_0 := false;
   AI_RAW_6005.___________0020_1 := false;
   AI_RAW_6005.RAW_MIN := 0;
   AI_RAW_6005.RAW_MAX := 27648;
   AI_RAW_6005.RAW_DESC := 'Resistance - 2-wire (6000 Ohm)';
   AI_RAW_6005.___________0030_1 := false;
   AI_RAW_6005.___________0030_2 := false;
   AI_RAW_6005.PARAM_TYPE := 16#06;
   AI_RAW_6005.PARAM_RANGE := 16#05;
   AI_RAW_6005.PARAM_COEF := 16#00;
   AI_RAW_6005.___________0040_1 := false;
   AI_RAW_6005.___________0040_2 := false;
   AI_RAW_6005.VALUE_COEF := 0.0;
   AI_RAW_600F.revInfo.REV_BLOCK := 'UT00801';
   AI_RAW_600F.revInfo.REV_NUMBER := '001.000';
   AI_RAW_600F.revInfo.REV_DATE := '2024-04-09';
   AI_RAW_600F.revInfo.REV_AUTHOR := 'M. Gledhill';
   AI_RAW_600F.___________0010_0 := false;
   AI_RAW_600F.___________0010_1 := false;
   AI_RAW_600F.AI_CODE := 16#600F;
   AI_RAW_600F.___________0020_0 := false;
   AI_RAW_600F.___________0020_1 := false;
   AI_RAW_600F.RAW_MIN := 0;
   AI_RAW_600F.RAW_MAX := 27648;
   AI_RAW_600F.RAW_DESC := 'Resistance - 2-wire (PTC)';
   AI_RAW_600F.___________0030_1 := false;
   AI_RAW_600F.___________0030_2 := false;
   AI_RAW_600F.PARAM_TYPE := 16#06;
   AI_RAW_600F.PARAM_RANGE := 16#0F;
   AI_RAW_600F.PARAM_COEF := 16#00;
   AI_RAW_600F.___________0040_1 := false;
   AI_RAW_600F.___________0040_2 := false;
   AI_RAW_600F.VALUE_COEF := 0.0;
   AI_RAW_7B0E.revInfo.REV_BLOCK := 'UT00801';
   AI_RAW_7B0E.revInfo.REV_NUMBER := '001.000';
   AI_RAW_7B0E.revInfo.REV_DATE := '2024-04-09';
   AI_RAW_7B0E.revInfo.REV_AUTHOR := 'M. Gledhill';
   AI_RAW_7B0E.___________0010_0 := false;
   AI_RAW_7B0E.___________0010_1 := false;
   AI_RAW_7B0E.AI_CODE := 16#7B0E;
   AI_RAW_7B0E.___________0020_0 := false;
   AI_RAW_7B0E.___________0020_1 := false;
   AI_RAW_7B0E.RAW_MIN := -5000;
   AI_RAW_7B0E.RAW_MAX := 15000;
   AI_RAW_7B0E.RAW_DESC := 'Thermal Resistance - 4-wire (Cu10 climate - 426)';
   AI_RAW_7B0E.___________0030_1 := false;
   AI_RAW_7B0E.___________0030_2 := false;
   AI_RAW_7B0E.PARAM_TYPE := 16#07;
   AI_RAW_7B0E.PARAM_RANGE := 16#0E;
   AI_RAW_7B0E.PARAM_COEF := 16#0B;
   AI_RAW_7B0E.___________0040_1 := false;
   AI_RAW_7B0E.___________0040_2 := false;
   AI_RAW_7B0E.VALUE_COEF := 0.00426;
   AI_RAW_7C0E.revInfo.REV_BLOCK := 'UT00801';
   AI_RAW_7C0E.revInfo.REV_NUMBER := '001.000';
   AI_RAW_7C0E.revInfo.REV_DATE := '2024-04-09';
   AI_RAW_7C0E.revInfo.REV_AUTHOR := 'M. Gledhill';
   AI_RAW_7C0E.___________0010_0 := false;
   AI_RAW_7C0E.___________0010_1 := false;
   AI_RAW_7C0E.AI_CODE := 16#7C0E;
   AI_RAW_7C0E.___________0020_0 := false;
   AI_RAW_7C0E.___________0020_1 := false;
   AI_RAW_7C0E.RAW_MIN := -5000;
   AI_RAW_7C0E.RAW_MAX := 15000;
   AI_RAW_7C0E.RAW_DESC := 'Thermal Resistance - 4-wire (Cu10 climate - 427)';
   AI_RAW_7C0E.___________0030_1 := false;
   AI_RAW_7C0E.___________0030_2 := false;
   AI_RAW_7C0E.PARAM_TYPE := 16#07;
   AI_RAW_7C0E.PARAM_RANGE := 16#0E;
   AI_RAW_7C0E.PARAM_COEF := 16#0C;
   AI_RAW_7C0E.___________0040_1 := false;
   AI_RAW_7C0E.___________0040_2 := false;
   AI_RAW_7C0E.VALUE_COEF := 0.00427;
   AI_RAW_7D0E.revInfo.REV_BLOCK := 'UT00801';
   AI_RAW_7D0E.revInfo.REV_NUMBER := '001.000';
   AI_RAW_7D0E.revInfo.REV_DATE := '2024-04-09';
   AI_RAW_7D0E.revInfo.REV_AUTHOR := 'M. Gledhill';
   AI_RAW_7D0E.___________0010_0 := false;
   AI_RAW_7D0E.___________0010_1 := false;
   AI_RAW_7D0E.AI_CODE := 16#7D0E;
   AI_RAW_7D0E.___________0020_0 := false;
   AI_RAW_7D0E.___________0020_1 := false;
   AI_RAW_7D0E.RAW_MIN := -5000;
   AI_RAW_7D0E.RAW_MAX := 15000;
   AI_RAW_7D0E.RAW_DESC := 'Thermal Resistance - 4-wire (Cu10 climate - 428)';
   AI_RAW_7D0E.___________0030_1 := false;
   AI_RAW_7D0E.___________0030_2 := false;
   AI_RAW_7D0E.PARAM_TYPE := 16#07;
   AI_RAW_7D0E.PARAM_RANGE := 16#0E;
   AI_RAW_7D0E.PARAM_COEF := 16#0D;
   AI_RAW_7D0E.___________0040_1 := false;
   AI_RAW_7D0E.___________0040_2 := false;
   AI_RAW_7D0E.VALUE_COEF := 0.00428;
   AI_RAW_7B0F.revInfo.REV_BLOCK := 'UT00801';
   AI_RAW_7B0F.revInfo.REV_NUMBER := '001.000';
   AI_RAW_7B0F.revInfo.REV_DATE := '2024-04-09';
   AI_RAW_7B0F.revInfo.REV_AUTHOR := 'M. Gledhill';
   AI_RAW_7B0F.___________0010_0 := false;
   AI_RAW_7B0F.___________0010_1 := false;
   AI_RAW_7B0F.AI_CODE := 16#7B0F;
   AI_RAW_7B0F.___________0020_0 := false;
   AI_RAW_7B0F.___________0020_1 := false;
   AI_RAW_7B0F.RAW_MIN := -500;
   AI_RAW_7B0F.RAW_MAX := 2000;
   AI_RAW_7B0F.RAW_DESC := 'Thermal Resistance - 4-wire (Cu10 standard - 426)';
   AI_RAW_7B0F.___________0030_1 := false;
   AI_RAW_7B0F.___________0030_2 := false;
   AI_RAW_7B0F.PARAM_TYPE := 16#07;
   AI_RAW_7B0F.PARAM_RANGE := 16#0F;
   AI_RAW_7B0F.PARAM_COEF := 16#0B;
   AI_RAW_7B0F.___________0040_1 := false;
   AI_RAW_7B0F.___________0040_2 := false;
   AI_RAW_7B0F.VALUE_COEF := 0.00426;
   AI_RAW_7C0F.revInfo.REV_BLOCK := 'UT00801';
   AI_RAW_7C0F.revInfo.REV_NUMBER := '001.000';
   AI_RAW_7C0F.revInfo.REV_DATE := '2024-04-09';
   AI_RAW_7C0F.revInfo.REV_AUTHOR := 'M. Gledhill';
   AI_RAW_7C0F.___________0010_0 := false;
   AI_RAW_7C0F.___________0010_1 := false;
   AI_RAW_7C0F.AI_CODE := 16#7C0F;
   AI_RAW_7C0F.___________0020_0 := false;
   AI_RAW_7C0F.___________0020_1 := false;
   AI_RAW_7C0F.RAW_MIN := -2000;
   AI_RAW_7C0F.RAW_MAX := 2600;
   AI_RAW_7C0F.RAW_DESC := 'Thermal Resistance - 4-wire (Cu10 standard - 427)';
   AI_RAW_7C0F.___________0030_1 := false;
   AI_RAW_7C0F.___________0030_2 := false;
   AI_RAW_7C0F.PARAM_TYPE := 16#07;
   AI_RAW_7C0F.PARAM_RANGE := 16#0F;
   AI_RAW_7C0F.PARAM_COEF := 16#0C;
   AI_RAW_7C0F.___________0040_1 := false;
   AI_RAW_7C0F.___________0040_2 := false;
   AI_RAW_7C0F.VALUE_COEF := 0.00427;
   AI_RAW_7D0F.revInfo.REV_BLOCK := 'UT00801';
   AI_RAW_7D0F.revInfo.REV_NUMBER := '001.000';
   AI_RAW_7D0F.revInfo.REV_DATE := '2024-04-09';
   AI_RAW_7D0F.revInfo.REV_AUTHOR := 'M. Gledhill';
   AI_RAW_7D0F.___________0010_0 := false;
   AI_RAW_7D0F.___________0010_1 := false;
   AI_RAW_7D0F.AI_CODE := 16#7D0F;
   AI_RAW_7D0F.___________0020_0 := false;
   AI_RAW_7D0F.___________0020_1 := false;
   AI_RAW_7D0F.RAW_MIN := -1800;
   AI_RAW_7D0F.RAW_MAX := 2000;
   AI_RAW_7D0F.RAW_DESC := 'Thermal Resistance - 4-wire (Cu10 standard - 428)';
   AI_RAW_7D0F.___________0030_1 := false;
   AI_RAW_7D0F.___________0030_2 := false;
   AI_RAW_7D0F.PARAM_TYPE := 16#07;
   AI_RAW_7D0F.PARAM_RANGE := 16#0F;
   AI_RAW_7D0F.PARAM_COEF := 16#0D;
   AI_RAW_7D0F.___________0040_1 := false;
   AI_RAW_7D0F.___________0040_2 := false;
   AI_RAW_7D0F.VALUE_COEF := 0.00428;
   AI_RAW_7B19.revInfo.REV_BLOCK := 'UT00801';
   AI_RAW_7B19.revInfo.REV_NUMBER := '001.000';
   AI_RAW_7B19.revInfo.REV_DATE := '2024-04-09';
   AI_RAW_7B19.revInfo.REV_AUTHOR := 'M. Gledhill';
   AI_RAW_7B19.___________0010_0 := false;
   AI_RAW_7B19.___________0010_1 := false;
   AI_RAW_7B19.AI_CODE := 16#7B19;
   AI_RAW_7B19.___________0020_0 := false;
   AI_RAW_7B19.___________0020_1 := false;
   AI_RAW_7B19.RAW_MIN := -5000;
   AI_RAW_7B19.RAW_MAX := 15000;
   AI_RAW_7B19.RAW_DESC := 'Thermal Resistance - 4-wire (Cu50 climate - 426)';
   AI_RAW_7B19.___________0030_1 := false;
   AI_RAW_7B19.___________0030_2 := false;
   AI_RAW_7B19.PARAM_TYPE := 16#07;
   AI_RAW_7B19.PARAM_RANGE := 16#19;
   AI_RAW_7B19.PARAM_COEF := 16#0B;
   AI_RAW_7B19.___________0040_1 := false;
   AI_RAW_7B19.___________0040_2 := false;
   AI_RAW_7B19.VALUE_COEF := 0.00426;
   AI_RAW_7C19.revInfo.REV_BLOCK := 'UT00801';
   AI_RAW_7C19.revInfo.REV_NUMBER := '001.000';
   AI_RAW_7C19.revInfo.REV_DATE := '2024-04-09';
   AI_RAW_7C19.revInfo.REV_AUTHOR := 'M. Gledhill';
   AI_RAW_7C19.___________0010_0 := false;
   AI_RAW_7C19.___________0010_1 := false;
   AI_RAW_7C19.AI_CODE := 16#7C19;
   AI_RAW_7C19.___________0020_0 := false;
   AI_RAW_7C19.___________0020_1 := false;
   AI_RAW_7C19.RAW_MIN := -5000;
   AI_RAW_7C19.RAW_MAX := 15000;
   AI_RAW_7C19.RAW_DESC := 'Thermal Resistance - 4-wire (Cu50 climate - 427)';
   AI_RAW_7C19.___________0030_1 := false;
   AI_RAW_7C19.___________0030_2 := false;
   AI_RAW_7C19.PARAM_TYPE := 16#07;
   AI_RAW_7C19.PARAM_RANGE := 16#19;
   AI_RAW_7C19.PARAM_COEF := 16#0C;
   AI_RAW_7C19.___________0040_1 := false;
   AI_RAW_7C19.___________0040_2 := false;
   AI_RAW_7C19.VALUE_COEF := 0.00427;
   AI_RAW_7D19.revInfo.REV_BLOCK := 'UT00801';
   AI_RAW_7D19.revInfo.REV_NUMBER := '001.000';
   AI_RAW_7D19.revInfo.REV_DATE := '2024-04-09';
   AI_RAW_7D19.revInfo.REV_AUTHOR := 'M. Gledhill';
   AI_RAW_7D19.___________0010_0 := false;
   AI_RAW_7D19.___________0010_1 := false;
   AI_RAW_7D19.AI_CODE := 16#7D19;
   AI_RAW_7D19.___________0020_0 := false;
   AI_RAW_7D19.___________0020_1 := false;
   AI_RAW_7D19.RAW_MIN := -5000;
   AI_RAW_7D19.RAW_MAX := 15000;
   AI_RAW_7D19.RAW_DESC := 'Thermal Resistance - 4-wire (Cu50 climate - 428)';
   AI_RAW_7D19.___________0030_1 := false;
   AI_RAW_7D19.___________0030_2 := false;
   AI_RAW_7D19.PARAM_TYPE := 16#07;
   AI_RAW_7D19.PARAM_RANGE := 16#19;
   AI_RAW_7D19.PARAM_COEF := 16#0D;
   AI_RAW_7D19.___________0040_1 := false;
   AI_RAW_7D19.___________0040_2 := false;
   AI_RAW_7D19.VALUE_COEF := 0.00428;
   AI_RAW_7B18.revInfo.REV_BLOCK := 'UT00801';
   AI_RAW_7B18.revInfo.REV_NUMBER := '001.000';
   AI_RAW_7B18.revInfo.REV_DATE := '2024-04-09';
   AI_RAW_7B18.revInfo.REV_AUTHOR := 'M. Gledhill';
   AI_RAW_7B18.___________0010_0 := false;
   AI_RAW_7B18.___________0010_1 := false;
   AI_RAW_7B18.AI_CODE := 16#7B18;
   AI_RAW_7B18.___________0020_0 := false;
   AI_RAW_7B18.___________0020_1 := false;
   AI_RAW_7B18.RAW_MIN := -500;
   AI_RAW_7B18.RAW_MAX := 2000;
   AI_RAW_7B18.RAW_DESC := 'Thermal Resistance - 4-wire (Cu50 standard - 426)';
   AI_RAW_7B18.___________0030_1 := false;
   AI_RAW_7B18.___________0030_2 := false;
   AI_RAW_7B18.PARAM_TYPE := 16#07;
   AI_RAW_7B18.PARAM_RANGE := 16#18;
   AI_RAW_7B18.PARAM_COEF := 16#0B;
   AI_RAW_7B18.___________0040_1 := false;
   AI_RAW_7B18.___________0040_2 := false;
   AI_RAW_7B18.VALUE_COEF := 0.00426;
   AI_RAW_7C18.revInfo.REV_BLOCK := 'UT00801';
   AI_RAW_7C18.revInfo.REV_NUMBER := '001.000';
   AI_RAW_7C18.revInfo.REV_DATE := '2024-04-09';
   AI_RAW_7C18.revInfo.REV_AUTHOR := 'M. Gledhill';
   AI_RAW_7C18.___________0010_0 := false;
   AI_RAW_7C18.___________0010_1 := false;
   AI_RAW_7C18.AI_CODE := 16#7C18;
   AI_RAW_7C18.___________0020_0 := false;
   AI_RAW_7C18.___________0020_1 := false;
   AI_RAW_7C18.RAW_MIN := -2000;
   AI_RAW_7C18.RAW_MAX := 2600;
   AI_RAW_7C18.RAW_DESC := 'Thermal Resistance - 4-wire (Cu50 standard - 427)';
   AI_RAW_7C18.___________0030_1 := false;
   AI_RAW_7C18.___________0030_2 := false;
   AI_RAW_7C18.PARAM_TYPE := 16#07;
   AI_RAW_7C18.PARAM_RANGE := 16#18;
   AI_RAW_7C18.PARAM_COEF := 16#0C;
   AI_RAW_7C18.___________0040_1 := false;
   AI_RAW_7C18.___________0040_2 := false;
   AI_RAW_7C18.VALUE_COEF := 0.00427;
   AI_RAW_7D18.revInfo.REV_BLOCK := 'UT00801';
   AI_RAW_7D18.revInfo.REV_NUMBER := '001.000';
   AI_RAW_7D18.revInfo.REV_DATE := '2024-04-09';
   AI_RAW_7D18.revInfo.REV_AUTHOR := 'M. Gledhill';
   AI_RAW_7D18.___________0010_0 := false;
   AI_RAW_7D18.___________0010_1 := false;
   AI_RAW_7D18.AI_CODE := 16#7D18;
   AI_RAW_7D18.___________0020_0 := false;
   AI_RAW_7D18.___________0020_1 := false;
   AI_RAW_7D18.RAW_MIN := -1800;
   AI_RAW_7D18.RAW_MAX := 2000;
   AI_RAW_7D18.RAW_DESC := 'Thermal Resistance - 4-wire (Cu50 standard - 428)';
   AI_RAW_7D18.___________0030_1 := false;
   AI_RAW_7D18.___________0030_2 := false;
   AI_RAW_7D18.PARAM_TYPE := 16#07;
   AI_RAW_7D18.PARAM_RANGE := 16#18;
   AI_RAW_7D18.PARAM_COEF := 16#0D;
   AI_RAW_7D18.___________0040_1 := false;
   AI_RAW_7D18.___________0040_2 := false;
   AI_RAW_7D18.VALUE_COEF := 0.00428;
   AI_RAW_7B1B.revInfo.REV_BLOCK := 'UT00801';
   AI_RAW_7B1B.revInfo.REV_NUMBER := '001.000';
   AI_RAW_7B1B.revInfo.REV_DATE := '2024-04-09';
   AI_RAW_7B1B.revInfo.REV_AUTHOR := 'M. Gledhill';
   AI_RAW_7B1B.___________0010_0 := false;
   AI_RAW_7B1B.___________0010_1 := false;
   AI_RAW_7B1B.AI_CODE := 16#7B1B;
   AI_RAW_7B1B.___________0020_0 := false;
   AI_RAW_7B1B.___________0020_1 := false;
   AI_RAW_7B1B.RAW_MIN := -5000;
   AI_RAW_7B1B.RAW_MAX := 15000;
   AI_RAW_7B1B.RAW_DESC := 'Thermal Resistance - 4-wire (Cu100 climate - 426)';
   AI_RAW_7B1B.___________0030_1 := false;
   AI_RAW_7B1B.___________0030_2 := false;
   AI_RAW_7B1B.PARAM_TYPE := 16#07;
   AI_RAW_7B1B.PARAM_RANGE := 16#1B;
   AI_RAW_7B1B.PARAM_COEF := 16#0B;
   AI_RAW_7B1B.___________0040_1 := false;
   AI_RAW_7B1B.___________0040_2 := false;
   AI_RAW_7B1B.VALUE_COEF := 0.00426;
   AI_RAW_7C1B.revInfo.REV_BLOCK := 'UT00801';
   AI_RAW_7C1B.revInfo.REV_NUMBER := '001.000';
   AI_RAW_7C1B.revInfo.REV_DATE := '2024-04-09';
   AI_RAW_7C1B.revInfo.REV_AUTHOR := 'M. Gledhill';
   AI_RAW_7C1B.___________0010_0 := false;
   AI_RAW_7C1B.___________0010_1 := false;
   AI_RAW_7C1B.AI_CODE := 16#7C1B;
   AI_RAW_7C1B.___________0020_0 := false;
   AI_RAW_7C1B.___________0020_1 := false;
   AI_RAW_7C1B.RAW_MIN := -5000;
   AI_RAW_7C1B.RAW_MAX := 15000;
   AI_RAW_7C1B.RAW_DESC := 'Thermal Resistance - 4-wire (Cu100 climate - 427)';
   AI_RAW_7C1B.___________0030_1 := false;
   AI_RAW_7C1B.___________0030_2 := false;
   AI_RAW_7C1B.PARAM_TYPE := 16#07;
   AI_RAW_7C1B.PARAM_RANGE := 16#1B;
   AI_RAW_7C1B.PARAM_COEF := 16#0C;
   AI_RAW_7C1B.___________0040_1 := false;
   AI_RAW_7C1B.___________0040_2 := false;
   AI_RAW_7C1B.VALUE_COEF := 0.00427;
   AI_RAW_7D1B.revInfo.REV_BLOCK := 'UT00801';
   AI_RAW_7D1B.revInfo.REV_NUMBER := '001.000';
   AI_RAW_7D1B.revInfo.REV_DATE := '2024-04-09';
   AI_RAW_7D1B.revInfo.REV_AUTHOR := 'M. Gledhill';
   AI_RAW_7D1B.___________0010_0 := false;
   AI_RAW_7D1B.___________0010_1 := false;
   AI_RAW_7D1B.AI_CODE := 16#7D1B;
   AI_RAW_7D1B.___________0020_0 := false;
   AI_RAW_7D1B.___________0020_1 := false;
   AI_RAW_7D1B.RAW_MIN := -5000;
   AI_RAW_7D1B.RAW_MAX := 15000;
   AI_RAW_7D1B.RAW_DESC := 'Thermal Resistance - 4-wire (Cu100 climate - 428)';
   AI_RAW_7D1B.___________0030_1 := false;
   AI_RAW_7D1B.___________0030_2 := false;
   AI_RAW_7D1B.PARAM_TYPE := 16#07;
   AI_RAW_7D1B.PARAM_RANGE := 16#1B;
   AI_RAW_7D1B.PARAM_COEF := 16#0D;
   AI_RAW_7D1B.___________0040_1 := false;
   AI_RAW_7D1B.___________0040_2 := false;
   AI_RAW_7D1B.VALUE_COEF := 0.00428;
   AI_RAW_7B1A.revInfo.REV_BLOCK := 'UT00801';
   AI_RAW_7B1A.revInfo.REV_NUMBER := '001.000';
   AI_RAW_7B1A.revInfo.REV_DATE := '2024-04-09';
   AI_RAW_7B1A.revInfo.REV_AUTHOR := 'M. Gledhill';
   AI_RAW_7B1A.___________0010_0 := false;
   AI_RAW_7B1A.___________0010_1 := false;
   AI_RAW_7B1A.AI_CODE := 16#7B1A;
   AI_RAW_7B1A.___________0020_0 := false;
   AI_RAW_7B1A.___________0020_1 := false;
   AI_RAW_7B1A.RAW_MIN := -500;
   AI_RAW_7B1A.RAW_MAX := 2000;
   AI_RAW_7B1A.RAW_DESC := 'Thermal Resistance - 4-wire (Cu100 standard - 426)';
   AI_RAW_7B1A.___________0030_1 := false;
   AI_RAW_7B1A.___________0030_2 := false;
   AI_RAW_7B1A.PARAM_TYPE := 16#07;
   AI_RAW_7B1A.PARAM_RANGE := 16#1A;
   AI_RAW_7B1A.PARAM_COEF := 16#0B;
   AI_RAW_7B1A.___________0040_1 := false;
   AI_RAW_7B1A.___________0040_2 := false;
   AI_RAW_7B1A.VALUE_COEF := 0.00426;
   AI_RAW_7C1A.revInfo.REV_BLOCK := 'UT00801';
   AI_RAW_7C1A.revInfo.REV_NUMBER := '001.000';
   AI_RAW_7C1A.revInfo.REV_DATE := '2024-04-09';
   AI_RAW_7C1A.revInfo.REV_AUTHOR := 'M. Gledhill';
   AI_RAW_7C1A.___________0010_0 := false;
   AI_RAW_7C1A.___________0010_1 := false;
   AI_RAW_7C1A.AI_CODE := 16#7C1A;
   AI_RAW_7C1A.___________0020_0 := false;
   AI_RAW_7C1A.___________0020_1 := false;
   AI_RAW_7C1A.RAW_MIN := -2000;
   AI_RAW_7C1A.RAW_MAX := 2600;
   AI_RAW_7C1A.RAW_DESC := 'Thermal Resistance - 4-wire (Cu100 standard - 427)';
   AI_RAW_7C1A.___________0030_1 := false;
   AI_RAW_7C1A.___________0030_2 := false;
   AI_RAW_7C1A.PARAM_TYPE := 16#07;
   AI_RAW_7C1A.PARAM_RANGE := 16#1A;
   AI_RAW_7C1A.PARAM_COEF := 16#0C;
   AI_RAW_7C1A.___________0040_1 := false;
   AI_RAW_7C1A.___________0040_2 := false;
   AI_RAW_7C1A.VALUE_COEF := 0.00427;
   AI_RAW_7D1A.revInfo.REV_BLOCK := 'UT00801';
   AI_RAW_7D1A.revInfo.REV_NUMBER := '001.000';
   AI_RAW_7D1A.revInfo.REV_DATE := '2024-04-09';
   AI_RAW_7D1A.revInfo.REV_AUTHOR := 'M. Gledhill';
   AI_RAW_7D1A.___________0010_0 := false;
   AI_RAW_7D1A.___________0010_1 := false;
   AI_RAW_7D1A.AI_CODE := 16#7D1A;
   AI_RAW_7D1A.___________0020_0 := false;
   AI_RAW_7D1A.___________0020_1 := false;
   AI_RAW_7D1A.RAW_MIN := -1800;
   AI_RAW_7D1A.RAW_MAX := 2000;
   AI_RAW_7D1A.RAW_DESC := 'Thermal Resistance - 4-wire (Cu100 standard - 428)';
   AI_RAW_7D1A.___________0030_1 := false;
   AI_RAW_7D1A.___________0030_2 := false;
   AI_RAW_7D1A.PARAM_TYPE := 16#07;
   AI_RAW_7D1A.PARAM_RANGE := 16#1A;
   AI_RAW_7D1A.PARAM_COEF := 16#0D;
   AI_RAW_7D1A.___________0040_1 := false;
   AI_RAW_7D1A.___________0040_2 := false;
   AI_RAW_7D1A.VALUE_COEF := 0.00428;
   AI_RAW_7A1D.revInfo.REV_BLOCK := 'UT00801';
   AI_RAW_7A1D.revInfo.REV_NUMBER := '001.000';
   AI_RAW_7A1D.revInfo.REV_DATE := '2024-04-09';
   AI_RAW_7A1D.revInfo.REV_AUTHOR := 'M. Gledhill';
   AI_RAW_7A1D.___________0010_0 := false;
   AI_RAW_7A1D.___________0010_1 := false;
   AI_RAW_7A1D.AI_CODE := 16#7A1D;
   AI_RAW_7A1D.___________0020_0 := false;
   AI_RAW_7A1D.___________0020_1 := false;
   AI_RAW_7A1D.RAW_MIN := -6000;
   AI_RAW_7A1D.RAW_MAX := 13000;
   AI_RAW_7A1D.RAW_DESC := 'Thermal Resistance - 4-wire (LG-Ni1000 climate - 500)';
   AI_RAW_7A1D.___________0030_1 := false;
   AI_RAW_7A1D.___________0030_2 := false;
   AI_RAW_7A1D.PARAM_TYPE := 16#07;
   AI_RAW_7A1D.PARAM_RANGE := 16#1D;
   AI_RAW_7A1D.PARAM_COEF := 16#0A;
   AI_RAW_7A1D.___________0040_1 := false;
   AI_RAW_7A1D.___________0040_2 := false;
   AI_RAW_7A1D.VALUE_COEF := 0.005;
   AI_RAW_7A1C.revInfo.REV_BLOCK := 'UT00801';
   AI_RAW_7A1C.revInfo.REV_NUMBER := '001.000';
   AI_RAW_7A1C.revInfo.REV_DATE := '2024-04-09';
   AI_RAW_7A1C.revInfo.REV_AUTHOR := 'M. Gledhill';
   AI_RAW_7A1C.___________0010_0 := false;
   AI_RAW_7A1C.___________0010_1 := false;
   AI_RAW_7A1C.AI_CODE := 16#7A1C;
   AI_RAW_7A1C.___________0020_0 := false;
   AI_RAW_7A1C.___________0020_1 := false;
   AI_RAW_7A1C.RAW_MIN := -600;
   AI_RAW_7A1C.RAW_MAX := 2500;
   AI_RAW_7A1C.RAW_DESC := 'Thermal Resistance - 4-wire (LG-Ni1000 standard - 500)';
   AI_RAW_7A1C.___________0030_1 := false;
   AI_RAW_7A1C.___________0030_2 := false;
   AI_RAW_7A1C.PARAM_TYPE := 16#07;
   AI_RAW_7A1C.PARAM_RANGE := 16#1C;
   AI_RAW_7A1C.PARAM_COEF := 16#0A;
   AI_RAW_7A1C.___________0040_1 := false;
   AI_RAW_7A1C.___________0040_2 := false;
   AI_RAW_7A1C.VALUE_COEF := 0.005;
   AI_RAW_771F.revInfo.REV_BLOCK := 'UT00801';
   AI_RAW_771F.revInfo.REV_NUMBER := '001.000';
   AI_RAW_771F.revInfo.REV_DATE := '2024-04-09';
   AI_RAW_771F.revInfo.REV_AUTHOR := 'M. Gledhill';
   AI_RAW_771F.___________0010_0 := false;
   AI_RAW_771F.___________0010_1 := false;
   AI_RAW_771F.AI_CODE := 16#771F;
   AI_RAW_771F.___________0020_0 := false;
   AI_RAW_771F.___________0020_1 := false;
   AI_RAW_771F.RAW_MIN := -6000;
   AI_RAW_771F.RAW_MAX := 13000;
   AI_RAW_771F.RAW_DESC := 'Thermal Resistance - 4-wire (Ni10 climate - 617)';
   AI_RAW_771F.___________0030_1 := false;
   AI_RAW_771F.___________0030_2 := false;
   AI_RAW_771F.PARAM_TYPE := 16#07;
   AI_RAW_771F.PARAM_RANGE := 16#1F;
   AI_RAW_771F.PARAM_COEF := 16#07;
   AI_RAW_771F.___________0040_1 := false;
   AI_RAW_771F.___________0040_2 := false;
   AI_RAW_771F.VALUE_COEF := 0.00617;
   AI_RAW_781F.revInfo.REV_BLOCK := 'UT00801';
   AI_RAW_781F.revInfo.REV_NUMBER := '001.000';
   AI_RAW_781F.revInfo.REV_DATE := '2024-04-09';
   AI_RAW_781F.revInfo.REV_AUTHOR := 'M. Gledhill';
   AI_RAW_781F.___________0010_0 := false;
   AI_RAW_781F.___________0010_1 := false;
   AI_RAW_781F.AI_CODE := 16#781F;
   AI_RAW_781F.___________0020_0 := false;
   AI_RAW_781F.___________0020_1 := false;
   AI_RAW_781F.RAW_MIN := -6000;
   AI_RAW_781F.RAW_MAX := 13000;
   AI_RAW_781F.RAW_DESC := 'Thermal Resistance - 4-wire (Ni10 climate - 618)';
   AI_RAW_781F.___________0030_1 := false;
   AI_RAW_781F.___________0030_2 := false;
   AI_RAW_781F.PARAM_TYPE := 16#07;
   AI_RAW_781F.PARAM_RANGE := 16#1F;
   AI_RAW_781F.PARAM_COEF := 16#08;
   AI_RAW_781F.___________0040_1 := false;
   AI_RAW_781F.___________0040_2 := false;
   AI_RAW_781F.VALUE_COEF := 0.00618;
   AI_RAW_791F.revInfo.REV_BLOCK := 'UT00801';
   AI_RAW_791F.revInfo.REV_NUMBER := '001.000';
   AI_RAW_791F.revInfo.REV_DATE := '2024-04-09';
   AI_RAW_791F.revInfo.REV_AUTHOR := 'M. Gledhill';
   AI_RAW_791F.___________0010_0 := false;
   AI_RAW_791F.___________0010_1 := false;
   AI_RAW_791F.AI_CODE := 16#791F;
   AI_RAW_791F.___________0020_0 := false;
   AI_RAW_791F.___________0020_1 := false;
   AI_RAW_791F.RAW_MIN := -6000;
   AI_RAW_791F.RAW_MAX := 13000;
   AI_RAW_791F.RAW_DESC := 'Thermal Resistance - 4-wire (Ni10 climate - 672)';
   AI_RAW_791F.___________0030_1 := false;
   AI_RAW_791F.___________0030_2 := false;
   AI_RAW_791F.PARAM_TYPE := 16#07;
   AI_RAW_791F.PARAM_RANGE := 16#1F;
   AI_RAW_791F.PARAM_COEF := 16#09;
   AI_RAW_791F.___________0040_1 := false;
   AI_RAW_791F.___________0040_2 := false;
   AI_RAW_791F.VALUE_COEF := 0.00672;
   AI_RAW_771E.revInfo.REV_BLOCK := 'UT00801';
   AI_RAW_771E.revInfo.REV_NUMBER := '001.000';
   AI_RAW_771E.revInfo.REV_DATE := '2024-04-09';
   AI_RAW_771E.revInfo.REV_AUTHOR := 'M. Gledhill';
   AI_RAW_771E.___________0010_0 := false;
   AI_RAW_771E.___________0010_1 := false;
   AI_RAW_771E.AI_CODE := 16#771E;
   AI_RAW_771E.___________0020_0 := false;
   AI_RAW_771E.___________0020_1 := false;
   AI_RAW_771E.RAW_MIN := -600;
   AI_RAW_771E.RAW_MAX := 1800;
   AI_RAW_771E.RAW_DESC := 'Thermal Resistance - 4-wire (Ni10 standard - 617)';
   AI_RAW_771E.___________0030_1 := false;
   AI_RAW_771E.___________0030_2 := false;
   AI_RAW_771E.PARAM_TYPE := 16#07;
   AI_RAW_771E.PARAM_RANGE := 16#1E;
   AI_RAW_771E.PARAM_COEF := 16#07;
   AI_RAW_771E.___________0040_1 := false;
   AI_RAW_771E.___________0040_2 := false;
   AI_RAW_771E.VALUE_COEF := 0.00617;
   AI_RAW_781E.revInfo.REV_BLOCK := 'UT00801';
   AI_RAW_781E.revInfo.REV_NUMBER := '001.000';
   AI_RAW_781E.revInfo.REV_DATE := '2024-04-09';
   AI_RAW_781E.revInfo.REV_AUTHOR := 'M. Gledhill';
   AI_RAW_781E.___________0010_0 := false;
   AI_RAW_781E.___________0010_1 := false;
   AI_RAW_781E.AI_CODE := 16#781E;
   AI_RAW_781E.___________0020_0 := false;
   AI_RAW_781E.___________0020_1 := false;
   AI_RAW_781E.RAW_MIN := -600;
   AI_RAW_781E.RAW_MAX := 2500;
   AI_RAW_781E.RAW_DESC := 'Thermal Resistance - 4-wire (Ni10 standard - 618)';
   AI_RAW_781E.___________0030_1 := false;
   AI_RAW_781E.___________0030_2 := false;
   AI_RAW_781E.PARAM_TYPE := 16#07;
   AI_RAW_781E.PARAM_RANGE := 16#1E;
   AI_RAW_781E.PARAM_COEF := 16#08;
   AI_RAW_781E.___________0040_1 := false;
   AI_RAW_781E.___________0040_2 := false;
   AI_RAW_781E.VALUE_COEF := 0.00618;
   AI_RAW_791E.revInfo.REV_BLOCK := 'UT00801';
   AI_RAW_791E.revInfo.REV_NUMBER := '001.000';
   AI_RAW_791E.revInfo.REV_DATE := '2024-04-09';
   AI_RAW_791E.revInfo.REV_AUTHOR := 'M. Gledhill';
   AI_RAW_791E.___________0010_0 := false;
   AI_RAW_791E.___________0010_1 := false;
   AI_RAW_791E.AI_CODE := 16#791E;
   AI_RAW_791E.___________0020_0 := false;
   AI_RAW_791E.___________0020_1 := false;
   AI_RAW_791E.RAW_MIN := -600;
   AI_RAW_791E.RAW_MAX := 2500;
   AI_RAW_791E.RAW_DESC := 'Thermal Resistance - 4-wire (Ni10 standard - 672)';
   AI_RAW_791E.___________0030_1 := false;
   AI_RAW_791E.___________0030_2 := false;
   AI_RAW_791E.PARAM_TYPE := 16#07;
   AI_RAW_791E.PARAM_RANGE := 16#1E;
   AI_RAW_791E.PARAM_COEF := 16#09;
   AI_RAW_791E.___________0040_1 := false;
   AI_RAW_791E.___________0040_2 := false;
   AI_RAW_791E.VALUE_COEF := 0.00672;
   AI_RAW_770D.revInfo.REV_BLOCK := 'UT00801';
   AI_RAW_770D.revInfo.REV_NUMBER := '001.000';
   AI_RAW_770D.revInfo.REV_DATE := '2024-04-09';
   AI_RAW_770D.revInfo.REV_AUTHOR := 'M. Gledhill';
   AI_RAW_770D.___________0010_0 := false;
   AI_RAW_770D.___________0010_1 := false;
   AI_RAW_770D.AI_CODE := 16#770D;
   AI_RAW_770D.___________0020_0 := false;
   AI_RAW_770D.___________0020_1 := false;
   AI_RAW_770D.RAW_MIN := -6000;
   AI_RAW_770D.RAW_MAX := 13000;
   AI_RAW_770D.RAW_DESC := 'Thermal Resistance - 4-wire (Ni120 climate - 617)';
   AI_RAW_770D.___________0030_1 := false;
   AI_RAW_770D.___________0030_2 := false;
   AI_RAW_770D.PARAM_TYPE := 16#07;
   AI_RAW_770D.PARAM_RANGE := 16#0D;
   AI_RAW_770D.PARAM_COEF := 16#07;
   AI_RAW_770D.___________0040_1 := false;
   AI_RAW_770D.___________0040_2 := false;
   AI_RAW_770D.VALUE_COEF := 0.00617;
   AI_RAW_780D.revInfo.REV_BLOCK := 'UT00801';
   AI_RAW_780D.revInfo.REV_NUMBER := '001.000';
   AI_RAW_780D.revInfo.REV_DATE := '2024-04-09';
   AI_RAW_780D.revInfo.REV_AUTHOR := 'M. Gledhill';
   AI_RAW_780D.___________0010_0 := false;
   AI_RAW_780D.___________0010_1 := false;
   AI_RAW_780D.AI_CODE := 16#780D;
   AI_RAW_780D.___________0020_0 := false;
   AI_RAW_780D.___________0020_1 := false;
   AI_RAW_780D.RAW_MIN := -6000;
   AI_RAW_780D.RAW_MAX := 13000;
   AI_RAW_780D.RAW_DESC := 'Thermal Resistance - 4-wire (Ni120 climate - 618)';
   AI_RAW_780D.___________0030_1 := false;
   AI_RAW_780D.___________0030_2 := false;
   AI_RAW_780D.PARAM_TYPE := 16#07;
   AI_RAW_780D.PARAM_RANGE := 16#0D;
   AI_RAW_780D.PARAM_COEF := 16#08;
   AI_RAW_780D.___________0040_1 := false;
   AI_RAW_780D.___________0040_2 := false;
   AI_RAW_780D.VALUE_COEF := 0.00618;
   AI_RAW_790D.revInfo.REV_BLOCK := 'UT00801';
   AI_RAW_790D.revInfo.REV_NUMBER := '001.000';
   AI_RAW_790D.revInfo.REV_DATE := '2024-04-09';
   AI_RAW_790D.revInfo.REV_AUTHOR := 'M. Gledhill';
   AI_RAW_790D.___________0010_0 := false;
   AI_RAW_790D.___________0010_1 := false;
   AI_RAW_790D.AI_CODE := 16#790D;
   AI_RAW_790D.___________0020_0 := false;
   AI_RAW_790D.___________0020_1 := false;
   AI_RAW_790D.RAW_MIN := -6000;
   AI_RAW_790D.RAW_MAX := 13000;
   AI_RAW_790D.RAW_DESC := 'Thermal Resistance - 4-wire (Ni120 climate - 672)';
   AI_RAW_790D.___________0030_1 := false;
   AI_RAW_790D.___________0030_2 := false;
   AI_RAW_790D.PARAM_TYPE := 16#07;
   AI_RAW_790D.PARAM_RANGE := 16#0D;
   AI_RAW_790D.PARAM_COEF := 16#09;
   AI_RAW_790D.___________0040_1 := false;
   AI_RAW_790D.___________0040_2 := false;
   AI_RAW_790D.VALUE_COEF := 0.00672;
   AI_RAW_770C.revInfo.REV_BLOCK := 'UT00801';
   AI_RAW_770C.revInfo.REV_NUMBER := '001.000';
   AI_RAW_770C.revInfo.REV_DATE := '2024-04-09';
   AI_RAW_770C.revInfo.REV_AUTHOR := 'M. Gledhill';
   AI_RAW_770C.___________0010_0 := false;
   AI_RAW_770C.___________0010_1 := false;
   AI_RAW_770C.AI_CODE := 16#770C;
   AI_RAW_770C.___________0020_0 := false;
   AI_RAW_770C.___________0020_1 := false;
   AI_RAW_770C.RAW_MIN := -600;
   AI_RAW_770C.RAW_MAX := 1800;
   AI_RAW_770C.RAW_DESC := 'Thermal Resistance - 4-wire (Ni120 standard - 617)';
   AI_RAW_770C.___________0030_1 := false;
   AI_RAW_770C.___________0030_2 := false;
   AI_RAW_770C.PARAM_TYPE := 16#07;
   AI_RAW_770C.PARAM_RANGE := 16#0C;
   AI_RAW_770C.PARAM_COEF := 16#07;
   AI_RAW_770C.___________0040_1 := false;
   AI_RAW_770C.___________0040_2 := false;
   AI_RAW_770C.VALUE_COEF := 0.00617;
   AI_RAW_780C.revInfo.REV_BLOCK := 'UT00801';
   AI_RAW_780C.revInfo.REV_NUMBER := '001.000';
   AI_RAW_780C.revInfo.REV_DATE := '2024-04-09';
   AI_RAW_780C.revInfo.REV_AUTHOR := 'M. Gledhill';
   AI_RAW_780C.___________0010_0 := false;
   AI_RAW_780C.___________0010_1 := false;
   AI_RAW_780C.AI_CODE := 16#780C;
   AI_RAW_780C.___________0020_0 := false;
   AI_RAW_780C.___________0020_1 := false;
   AI_RAW_780C.RAW_MIN := -600;
   AI_RAW_780C.RAW_MAX := 2500;
   AI_RAW_780C.RAW_DESC := 'Thermal Resistance - 4-wire (Ni120 standard - 618)';
   AI_RAW_780C.___________0030_1 := false;
   AI_RAW_780C.___________0030_2 := false;
   AI_RAW_780C.PARAM_TYPE := 16#07;
   AI_RAW_780C.PARAM_RANGE := 16#0C;
   AI_RAW_780C.PARAM_COEF := 16#08;
   AI_RAW_780C.___________0040_1 := false;
   AI_RAW_780C.___________0040_2 := false;
   AI_RAW_780C.VALUE_COEF := 0.00618;
   AI_RAW_790C.revInfo.REV_BLOCK := 'UT00801';
   AI_RAW_790C.revInfo.REV_NUMBER := '001.000';
   AI_RAW_790C.revInfo.REV_DATE := '2024-04-09';
   AI_RAW_790C.revInfo.REV_AUTHOR := 'M. Gledhill';
   AI_RAW_790C.___________0010_0 := false;
   AI_RAW_790C.___________0010_1 := false;
   AI_RAW_790C.AI_CODE := 16#790C;
   AI_RAW_790C.___________0020_0 := false;
   AI_RAW_790C.___________0020_1 := false;
   AI_RAW_790C.RAW_MIN := -600;
   AI_RAW_790C.RAW_MAX := 2500;
   AI_RAW_790C.RAW_DESC := 'Thermal Resistance - 4-wire (Ni120 standard - 672)';
   AI_RAW_790C.___________0030_1 := false;
   AI_RAW_790C.___________0030_2 := false;
   AI_RAW_790C.PARAM_TYPE := 16#07;
   AI_RAW_790C.PARAM_RANGE := 16#0C;
   AI_RAW_790C.PARAM_COEF := 16#09;
   AI_RAW_790C.___________0040_1 := false;
   AI_RAW_790C.___________0040_2 := false;
   AI_RAW_790C.VALUE_COEF := 0.00672;
   AI_RAW_7701.revInfo.REV_BLOCK := 'UT00801';
   AI_RAW_7701.revInfo.REV_NUMBER := '001.000';
   AI_RAW_7701.revInfo.REV_DATE := '2024-04-09';
   AI_RAW_7701.revInfo.REV_AUTHOR := 'M. Gledhill';
   AI_RAW_7701.___________0010_0 := false;
   AI_RAW_7701.___________0010_1 := false;
   AI_RAW_7701.AI_CODE := 16#7701;
   AI_RAW_7701.___________0020_0 := false;
   AI_RAW_7701.___________0020_1 := false;
   AI_RAW_7701.RAW_MIN := -6000;
   AI_RAW_7701.RAW_MAX := 13000;
   AI_RAW_7701.RAW_DESC := 'Thermal Resistance - 4-wire (Ni100 climate - 617)';
   AI_RAW_7701.___________0030_1 := false;
   AI_RAW_7701.___________0030_2 := false;
   AI_RAW_7701.PARAM_TYPE := 16#07;
   AI_RAW_7701.PARAM_RANGE := 16#01;
   AI_RAW_7701.PARAM_COEF := 16#07;
   AI_RAW_7701.___________0040_1 := false;
   AI_RAW_7701.___________0040_2 := false;
   AI_RAW_7701.VALUE_COEF := 0.00617;
   AI_RAW_7801.revInfo.REV_BLOCK := 'UT00801';
   AI_RAW_7801.revInfo.REV_NUMBER := '001.000';
   AI_RAW_7801.revInfo.REV_DATE := '2024-04-09';
   AI_RAW_7801.revInfo.REV_AUTHOR := 'M. Gledhill';
   AI_RAW_7801.___________0010_0 := false;
   AI_RAW_7801.___________0010_1 := false;
   AI_RAW_7801.AI_CODE := 16#7801;
   AI_RAW_7801.___________0020_0 := false;
